LIN {X 0,Y 389.238,Z 288.654,A -85,B 0,C 180,E1 -14313.105,E2 -14313.105} C_VEL
LIN {X 0,Y 387.614,Z 288.058,A -85,B 0,C 180,E1 -14314.941,E2 -14314.941} C_VEL
LIN {X 0,Y 385.469,Z 286.733,A -85,B 0,C 180,E1 -14316.684,E2 -14316.684} C_VEL
LIN {X 0,Y 383.225,Z 284.713,A -85,B 0,C 180,E1 -14318.163,E2 -14318.163} C_VEL
LIN {X 0,Y 380.545,Z 281.669,A -85,B 0,C 180,E1 -14319.669,E2 -14319.669} C_VEL
LIN {X 0,Y 377.534,Z 279.906,A -85,B 0,C 180,E1 -14321.039,E2 -14321.039} C_VEL
LIN {X 0,Y 374.063,Z 276.681,A -85,B 0,C 180,E1 -14322.478,E2 -14322.478} C_VEL
LIN {X 0,Y 371.999,Z 274.442,A -85,B 0,C 180,E1 -14323.274,E2 -14323.274} C_VEL
LIN {X 0,Y 368.238,Z 271.447,A -85,B 0,C 180,E1 -14324.55,E2 -14324.55} C_VEL
LIN {X 0,Y 365.07,Z 267.86,A -85,B 0,C 180,E1 -14325.587,E2 -14325.587} C_VEL
LIN {X 0,Y 361.353,Z 264.675,A -85,B 0,C 180,E1 -14326.692,E2 -14326.692} C_VEL
LIN {X 0,Y 358.552,Z 261.44,A -85,B 0,C 180,E1 -14327.482,E2 -14327.482} C_VEL
LIN {X 0,Y 355.376,Z 258.454,A -85,B 0,C 180,E1 -14328.333,E2 -14328.333} C_VEL
LIN {X 0,Y 353.051,Z 255.522,A -85,B 0,C 180,E1 -14328.94,E2 -14328.94} C_VEL
LIN {X 0,Y 350.001,Z 252.371,A -85,B 0,C 180,E1 -14329.706,E2 -14329.706} C_VEL
LIN {X 0,Y 348.215,Z 249.968,A -85,B 0,C 180,E1 -14330.137,E2 -14330.137} C_VEL
LIN {X 0,Y 345.498,Z 247.058,A -85,B 0,C 180,E1 -14330.785,E2 -14330.785} C_VEL
LIN {X 0,Y 344.015,Z 244.683,A -85,B 0,C 180,E1 -14331.145,E2 -14331.145} C_VEL
LIN {X 0,Y 341.721,Z 242.357,A -85,B 0,C 180,E1 -14331.634,E2 -14331.634} C_VEL
LIN {X 0,Y 340.82,Z 240.079,A -85,B 0,C 180,E1 -14331.984,E2 -14331.984} C_VEL
LIN {X 0,Y 340.743,Z 239.555,A -85,B 0,C 180,E1 -14332.43,E2 -14332.43} C_VEL
LIN {X 0,Y 340.769,Z 239.539,A -85,B 0,C 180,E1 -14335.665,E2 -14335.665} C_VEL
LIN {X 0,Y 340.724,Z 239.527,A -85,B 0,C 180,E1 -14338.321,E2 -14338.321} C_VEL
LIN {X 0,Y 340.694,Z 239.543,A -85,B 0,C 180,E1 -14341.045,E2 -14341.045} C_VEL
LIN {X 0,Y 340.714,Z 239.518,A -85,B 0,C 180,E1 -14345.279,E2 -14345.279} C_VEL
LIN {X 0,Y 340.714,Z 239.545,A -85,B 0,C 180,E1 -14348.388,E2 -14348.388} C_VEL
LIN {X 0,Y 340.702,Z 239.5,A -85,B 0,C 180,E1 -14352.047,E2 -14352.047} C_VEL
LIN {X 0,Y 340.751,Z 239.541,A -85,B 0,C 180,E1 -14356.209,E2 -14356.209} C_VEL
LIN {X 0,Y 340.761,Z 239.524,A -85,B 0,C 180,E1 -14359.738,E2 -14359.738} C_VEL
LIN {X 0,Y 340.708,Z 239.542,A -85,B 0,C 180,E1 -14363.56,E2 -14363.56} C_VEL
LIN {X 0,Y 340.689,Z 239.532,A -85,B 0,C 180,E1 -14366.154,E2 -14366.154} C_VEL
LIN {X 0,Y 340.772,Z 239.531,A -85,B 0,C 180,E1 -14370.333,E2 -14370.333} C_VEL
LIN {X 0,Y 340.801,Z 239.508,A -85,B 0,C 180,E1 -14373.021,E2 -14373.021} C_VEL
LIN {X 0,Y 340.758,Z 239.53,A -85,B 0,C 180,E1 -14374.684,E2 -14374.684} C_VEL
LIN {X 0,Y 340.074,Z 239.623,A -85,B 0,C 180,E1 -14375.671,E2 -14375.671} C_VEL
LIN {X 0,Y 337.177,Z 239.985,A -85,B 0,C 180,E1 -14377.275,E2 -14377.275} C_VEL
LIN {X 0,Y 334.754,Z 240.278,A -85,B 0,C 180,E1 -14378.574,E2 -14378.574} C_VEL
LIN {X 0,Y 333.754,Z 240.389,A -85,B 0,C 180,E1 -14379.58,E2 -14379.58} C_VEL
LIN {X 0,Y 333.694,Z 240.393,A -85,B 0,C 180,E1 -14379.921,E2 -14379.921} C_VEL
LIN {X 0,Y 333.745,Z 240.399,A -85,B 0,C 180,E1 -14382.854,E2 -14382.854} C_VEL
LIN {X 0,Y 333.795,Z 240.402,A -85,B 0,C 180,E1 -14386.609,E2 -14386.609} C_VEL
LIN {X 0,Y 333.849,Z 240.365,A -85,B 0,C 180,E1 -14390.305,E2 -14390.305} C_VEL
LIN {X 0,Y 334.004,Z 240.369,A -85,B 0,C 180,E1 -14392.748,E2 -14392.748} C_VEL
LIN {X 0,Y 333.808,Z 240.407,A -85,B 0,C 180,E1 -14395.17,E2 -14395.17} C_VEL
LIN {X 0,Y 334.106,Z 240.351,A -85,B 0,C 180,E1 -14397.589,E2 -14397.589} C_VEL
LIN {X 0,Y 334.226,Z 240.318,A -85,B 0,C 180,E1 -14400.001,E2 -14400.001} C_VEL
LIN {X 0,Y 334.105,Z 240.356,A -85,B 0,C 180,E1 -14402.412,E2 -14402.412} C_VEL
LIN {X 0,Y 333.998,Z 240.376,A -85,B 0,C 180,E1 -14406.04,E2 -14406.04} C_VEL
LIN {X 0,Y 333.82,Z 240.368,A -85,B 0,C 180,E1 -14409.697,E2 -14409.697} C_VEL
LIN {X 0,Y 333.797,Z 240.403,A -85,B 0,C 180,E1 -14413.392,E2 -14413.392} C_VEL
LIN {X 0,Y 333.719,Z 240.394,A -85,B 0,C 180,E1 -14417.148,E2 -14417.148} C_VEL
LIN {X 0,Y 333.719,Z 240.392,A -85,B 0,C 180,E1 -14419.692,E2 -14419.692} C_VEL
LIN {X 0,Y 333.692,Z 240.415,A -85,B 0,C 180,E1 -14422.279,E2 -14422.279} C_VEL
LIN {X 0,Y 333.735,Z 240.391,A -85,B 0,C 180,E1 -14426.247,E2 -14426.247} C_VEL
LIN {X 0,Y 333.691,Z 240.412,A -85,B 0,C 180,E1 -14428.975,E2 -14428.975} C_VEL
LIN {X 0,Y 333.644,Z 240.414,A -85,B 0,C 180,E1 -14432.587,E2 -14432.587} C_VEL
LIN {X 0,Y 333.675,Z 240.415,A -85,B 0,C 180,E1 -14436.14,E2 -14436.14} C_VEL
LIN {X 0,Y 333.648,Z 240.414,A -85,B 0,C 180,E1 -14439.193,E2 -14439.193} C_VEL
LIN {X 0,Y 333.634,Z 240.428,A -85,B 0,C 180,E1 -14442.501,E2 -14442.501} C_VEL
LIN {X 0,Y 333.598,Z 240.43,A -85,B 0,C 180,E1 -14445.956,E2 -14445.956} C_VEL
LIN {X 0,Y 333.649,Z 240.398,A -85,B 0,C 180,E1 -14449.316,E2 -14449.316} C_VEL
LIN {X 0,Y 333.667,Z 240.415,A -85,B 0,C 180,E1 -14453.168,E2 -14453.168} C_VEL
LIN {X 0,Y 333.701,Z 240.526,A -85,B 0,C 180,E1 -14456.885,E2 -14456.885} C_VEL
LIN {X 0,Y 335.005,Z 246.874,A -85,B 0,C 180,E1 -14459.332,E2 -14459.332} C_VEL
LIN {X 0,Y 336.843,Z 256.44,A -85,B 0,C 180,E1 -14462.677,E2 -14462.677} C_VEL
LIN {X 0,Y 337.125,Z 259.361,A -85,B 0,C 180,E1 -14463.692,E2 -14463.692} C_VEL
LIN {X 0,Y 336.268,Z 266.228,A -85,B 0,C 180,E1 -14465.913,E2 -14465.913} C_VEL
LIN {X 0,Y 336.94,Z 270.047,A -85,B 0,C 180,E1 -14466.119,E2 -14466.119} C_VEL
LIN {X 0,Y 341.597,Z 292.634,A -85,B 0,C 180,E1 -14466.967,E2 -14466.967} C_VEL
LIN {X 0,Y 343.681,Z 305.633,A -85,B 0,C 180,E1 -14467.402,E2 -14467.402} C_VEL
LIN {X 0,Y 342.412,Z 371.156,A -85,B 0,C 180,E1 -14468.792,E2 -14468.792} C_VEL
LIN {X 0,Y 341.886,Z 381.9,A -85,B 0,C 180,E1 -14469.152,E2 -14469.152} C_VEL
LIN {X 0,Y 341.255,Z 391.001,A -85,B 0,C 180,E1 -14469.585,E2 -14469.585} C_VEL
LIN {X 0,Y 340.336,Z 401.361,A -85,B 0,C 180,E1 -14470.236,E2 -14470.236} C_VEL
LIN {X 0,Y 339.44,Z 410.495,A -85,B 0,C 180,E1 -14470.968,E2 -14470.968} C_VEL
LIN {X 0,Y 338.419,Z 419.49,A -85,B 0,C 180,E1 -14471.85,E2 -14471.85} C_VEL
LIN {X 0,Y 337.282,Z 428.216,A -85,B 0,C 180,E1 -14472.883,E2 -14472.883} C_VEL
LIN {X 0,Y 336.343,Z 435.977,A -85,B 0,C 180,E1 -14473.986,E2 -14473.986} C_VEL
LIN {X 0,Y 335.454,Z 442.832,A -85,B 0,C 180,E1 -14475.129,E2 -14475.129} C_VEL
LIN {X 0,Y 334.667,Z 449.035,A -85,B 0,C 180,E1 -14476.335,E2 -14476.335} C_VEL
LIN {X 0,Y 333.732,Z 455.57,A -85,B 0,C 180,E1 -14477.843,E2 -14477.843} C_VEL
LIN {X 0,Y 333.236,Z 460.074,A -85,B 0,C 180,E1 -14479.058,E2 -14479.058} C_VEL
LIN {X 0,Y 332.605,Z 465.566,A -85,B 0,C 180,E1 -14480.882,E2 -14480.882} C_VEL
LIN {X 0,Y 332.202,Z 469.891,A -85,B 0,C 180,E1 -14482.708,E2 -14482.708} C_VEL
LIN {X 0,Y 332.034,Z 472.629,A -85,B 0,C 180,E1 -14484.174,E2 -14484.174} C_VEL
LIN {X 0,Y 331.97,Z 475.448,A -85,B 0,C 180,E1 -14486.359,E2 -14486.359} C_VEL
LIN {X 0,Y 331.916,Z 476.506,A -85,B 0,C 180,E1 -14487.573,E2 -14487.573} C_VEL
LIN {X 0,Y 331.913,Z 477.095,A -85,B 0,C 180,E1 -14488.787,E2 -14488.787} C_VEL
LIN {X 0,Y 331.913,Z 477.095,A -85,B 0,C 180,E1 -14491.213,E2 -14491.213} C_VEL
LIN {X 0,Y 331.916,Z 476.506,A -85,B 0,C 180,E1 -14492.427,E2 -14492.427} C_VEL
LIN {X 0,Y 331.971,Z 474.059,A -85,B 0,C 180,E1 -14494.858,E2 -14494.858} C_VEL
LIN {X 0,Y 332.105,Z 471.109,A -85,B 0,C 180,E1 -14496.684,E2 -14496.684} C_VEL
LIN {X 0,Y 332.461,Z 467.12,A -85,B 0,C 180,E1 -14498.51,E2 -14498.51} C_VEL
LIN {X 0,Y 332.985,Z 461.99,A -85,B 0,C 180,E1 -14500.335,E2 -14500.335} C_VEL
LIN {X 0,Y 333.589,Z 456.726,A -85,B 0,C 180,E1 -14501.854,E2 -14501.854} C_VEL
LIN {X 0,Y 334.455,Z 450.41,A -85,B 0,C 180,E1 -14503.364,E2 -14503.364} C_VEL
LIN {X 0,Y 335.208,Z 444.458,A -85,B 0,C 180,E1 -14504.572,E2 -14504.572} C_VEL
LIN {X 0,Y 336.147,Z 437.531,A -85,B 0,C 180,E1 -14505.771,E2 -14505.771} C_VEL
LIN {X 0,Y 337.155,Z 429.351,A -85,B 0,C 180,E1 -14506.967,E2 -14506.967} C_VEL
LIN {X 0,Y 338.249,Z 420.841,A -85,B 0,C 180,E1 -14508.003,E2 -14508.003} C_VEL
LIN {X 0,Y 339.26,Z 412.127,A -85,B 0,C 180,E1 -14508.886,E2 -14508.886} C_VEL
LIN {X 0,Y 340.256,Z 402.369,A -85,B 0,C 180,E1 -14509.69,E2 -14509.69} C_VEL
LIN {X 0,Y 341.184,Z 392.289,A -85,B 0,C 180,E1 -14510.341,E2 -14510.341} C_VEL
LIN {X 0,Y 341.848,Z 382.775,A -85,B 0,C 180,E1 -14510.811,E2 -14510.811} C_VEL
LIN {X 0,Y 342.38,Z 372.463,A -85,B 0,C 180,E1 -14511.17,E2 -14511.17} C_VEL
LIN {X 0,Y 343.694,Z 305.784,A -85,B 0,C 180,E1 -14512.594,E2 -14512.594} C_VEL
LIN {X 0,Y 339.925,Z 283.944,A -85,B 0,C 180,E1 -14513.347,E2 -14513.347} C_VEL
LIN {X 0,Y 336.278,Z 266.684,A -85,B 0,C 180,E1 -14514.03,E2 -14514.03} C_VEL
LIN {X 0,Y 336.36,Z 265.08,A -85,B 0,C 180,E1 -14514.405,E2 -14514.405} C_VEL
LIN {X 0,Y 337.108,Z 259.382,A -85,B 0,C 180,E1 -14516.302,E2 -14516.302} C_VEL
LIN {X 0,Y 336.549,Z 254.647,A -85,B 0,C 180,E1 -14517.961,E2 -14517.961} C_VEL
LIN {X 0,Y 334.535,Z 244.335,A -85,B 0,C 180,E1 -14521.682,E2 -14521.682} C_VEL
LIN {X 0,Y 333.674,Z 240.436,A -85,B 0,C 180,E1 -14523.204,E2 -14523.204} C_VEL
LIN {X 0,Y 333.667,Z 240.415,A -85,B 0,C 180,E1 -14526.832,E2 -14526.832} C_VEL
LIN {X 0,Y 333.648,Z 240.398,A -85,B 0,C 180,E1 -14530.767,E2 -14530.767} C_VEL
LIN {X 0,Y 333.595,Z 240.428,A -85,B 0,C 180,E1 -14534.25,E2 -14534.25} C_VEL
LIN {X 0,Y 333.643,Z 240.428,A -85,B 0,C 180,E1 -14537.618,E2 -14537.618} C_VEL
LIN {X 0,Y 333.653,Z 240.416,A -85,B 0,C 180,E1 -14541.202,E2 -14541.202} C_VEL
LIN {X 0,Y 333.675,Z 240.415,A -85,B 0,C 180,E1 -14543.86,E2 -14543.86} C_VEL
LIN {X 0,Y 333.644,Z 240.414,A -85,B 0,C 180,E1 -14547.413,E2 -14547.413} C_VEL
LIN {X 0,Y 333.691,Z 240.412,A -85,B 0,C 180,E1 -14551.025,E2 -14551.025} C_VEL
LIN {X 0,Y 333.735,Z 240.391,A -85,B 0,C 180,E1 -14553.753,E2 -14553.753} C_VEL
LIN {X 0,Y 333.72,Z 240.41,A -85,B 0,C 180,E1 -14557.913,E2 -14557.913} C_VEL
LIN {X 0,Y 333.741,Z 240.382,A -85,B 0,C 180,E1 -14561.586,E2 -14561.586} C_VEL
LIN {X 0,Y 333.808,Z 240.402,A -85,B 0,C 180,E1 -14565.576,E2 -14565.576} C_VEL
LIN {X 0,Y 333.817,Z 240.377,A -85,B 0,C 180,E1 -14569.077,E2 -14569.077} C_VEL
LIN {X 0,Y 333.968,Z 240.369,A -85,B 0,C 180,E1 -14572.746,E2 -14572.746} C_VEL
LIN {X 0,Y 333.804,Z 240.406,A -85,B 0,C 180,E1 -14575.168,E2 -14575.168} C_VEL
LIN {X 0,Y 334.105,Z 240.356,A -85,B 0,C 180,E1 -14577.588,E2 -14577.588} C_VEL
LIN {X 0,Y 334.226,Z 240.318,A -85,B 0,C 180,E1 -14579.999,E2 -14579.999} C_VEL
LIN {X 0,Y 334.106,Z 240.351,A -85,B 0,C 180,E1 -14582.411,E2 -14582.411} C_VEL
LIN {X 0,Y 333.99,Z 240.374,A -85,B 0,C 180,E1 -14586.597,E2 -14586.597} C_VEL
LIN {X 0,Y 333.849,Z 240.365,A -85,B 0,C 180,E1 -14589.695,E2 -14589.695} C_VEL
LIN {X 0,Y 333.795,Z 240.402,A -85,B 0,C 180,E1 -14593.391,E2 -14593.391} C_VEL
LIN {X 0,Y 333.745,Z 240.399,A -85,B 0,C 180,E1 -14597.146,E2 -14597.146} C_VEL
LIN {X 0,Y 333.729,Z 240.386,A -85,B 0,C 180,E1 -14599.69,E2 -14599.69} C_VEL
LIN {X 0,Y 333.667,Z 240.421,A -85,B 0,C 180,E1 -14603.59,E2 -14603.59} C_VEL
LIN {X 0,Y 333.732,Z 240.394,A -85,B 0,C 180,E1 -14606.246,E2 -14606.246} C_VEL
LIN {X 0,Y 333.708,Z 240.407,A -85,B 0,C 180,E1 -14608.972,E2 -14608.972} C_VEL
LIN {X 0,Y 333.64,Z 240.419,A -85,B 0,C 180,E1 -14612.586,E2 -14612.586} C_VEL
LIN {X 0,Y 333.673,Z 240.413,A -85,B 0,C 180,E1 -14616.138,E2 -14616.138} C_VEL
LIN {X 0,Y 333.679,Z 240.417,A -85,B 0,C 180,E1 -14619.187,E2 -14619.187} C_VEL
LIN {X 0,Y 333.7,Z 240.418,A -85,B 0,C 180,E1 -14622.513,E2 -14622.513} C_VEL
LIN {X 0,Y 333.631,Z 240.402,A -85,B 0,C 180,E1 -14625.961,E2 -14625.961} C_VEL
LIN {X 0,Y 333.651,Z 240.389,A -85,B 0,C 180,E1 -14629.314,E2 -14629.314} C_VEL
LIN {X 0,Y 333.652,Z 240.424,A -85,B 0,C 180,E1 -14632.349,E2 -14632.349} C_VEL
LIN {X 0,Y 333.67,Z 240.392,A -85,B 0,C 180,E1 -14635.341,E2 -14635.341} C_VEL
LIN {X 0,Y 333.686,Z 240.404,A -85,B 0,C 180,E1 -14639.637,E2 -14639.637} C_VEL
LIN {X 0,Y 333.736,Z 240.41,A -85,B 0,C 180,E1 -14642.401,E2 -14642.401} C_VEL
LIN {X 0,Y 333.723,Z 240.417,A -85,B 0,C 180,E1 -14645.091,E2 -14645.091} C_VEL
LIN {X 0,Y 333.714,Z 240.563,A -85,B 0,C 180,E1 -14646.635,E2 -14646.635} C_VEL
LIN {X 0,Y 333.902,Z 241.475,A -85,B 0,C 180,E1 -14646.906,E2 -14646.906} C_VEL
LIN {X 0,Y 335.441,Z 244.25,A -85,B 0,C 180,E1 -14647.293,E2 -14647.293} C_VEL
LIN {X 0,Y 337.24,Z 246.138,A -85,B 0,C 180,E1 -14647.649,E2 -14647.649} C_VEL
LIN {X 0,Y 339.606,Z 249.544,A -85,B 0,C 180,E1 -14648.193,E2 -14648.193} C_VEL
LIN {X 0,Y 341.244,Z 251.3,A -85,B 0,C 180,E1 -14648.55,E2 -14648.55} C_VEL
LIN {X 0,Y 344.183,Z 255.015,A -85,B 0,C 180,E1 -14649.205,E2 -14649.205} C_VEL
LIN {X 0,Y 346.131,Z 257.085,A -85,B 0,C 180,E1 -14649.669,E2 -14649.669} C_VEL
LIN {X 0,Y 349.255,Z 260.734,A -85,B 0,C 180,E1 -14650.409,E2 -14650.409} C_VEL
LIN {X 0,Y 351.306,Z 262.788,A -85,B 0,C 180,E1 -14650.915,E2 -14650.915} C_VEL
LIN {X 0,Y 354.984,Z 266.845,A -85,B 0,C 180,E1 -14651.859,E2 -14651.859} C_VEL
LIN {X 0,Y 357.12,Z 268.84,A -85,B 0,C 180,E1 -14652.431,E2 -14652.431} C_VEL
LIN {X 0,Y 361.088,Z 272.942,A -85,B 0,C 180,E1 -14653.544,E2 -14653.544} C_VEL
LIN {X 0,Y 363.916,Z 275.38,A -85,B 0,C 180,E1 -14654.391,E2 -14654.391} C_VEL
LIN {X 0,Y 367.522,Z 279.123,A -85,B 0,C 180,E1 -14655.553,E2 -14655.553} C_VEL
LIN {X 0,Y 371.229,Z 282.06,A -85,B 0,C 180,E1 -14656.813,E2 -14656.813} C_VEL
LIN {X 0,Y 374.888,Z 285.747,A -85,B 0,C 180,E1 -14658.242,E2 -14658.242} C_VEL
LIN {X 0,Y 378.477,Z 288.218,A -85,B 0,C 180,E1 -14659.786,E2 -14659.786} C_VEL
LIN {X 0,Y 379.883,Z 289.155,A -85,B 0,C 180,E1 -14660.464,E2 -14660.464} C_VEL
LIN {X 0,Y 382.521,Z 292.118,A -85,B 0,C 180,E1 -14661.961,E2 -14661.961} C_VEL
LIN {X 0,Y 384.968,Z 294.058,A -85,B 0,C 180,E1 -14663.58,E2 -14663.58} C_VEL
LIN {X 0,Y 387.283,Z 295.335,A -85,B 0,C 180,E1 -14665.578,E2 -14665.578} C_VEL
LIN {X 0,Y 388.665,Z 295.823,A -85,B 0,C 180,E1 -14667.428,E2 -14667.428} C_VEL
LIN {X 0,Y 389.239,Z 296.26,A -85,B 0,C 180,E1 -14668.965,E2 -14668.965} C_VEL
LIN {X 0,Y 389.407,Z 296.18,A -85,B 0,C 180,E1 -14670,E2 -14670} C_VEL
LIN {X 0,Y 389.127,Z 296.134,A -85,B 0,C 180,E1 -14671.552,E2 -14671.552} C_VEL
LIN {X 0,Y 388.361,Z 295.7,A -85,B 0,C 180,E1 -14673.112,E2 -14673.112} C_VEL
LIN {X 0,Y 386.736,Z 295.097,A -85,B 0,C 180,E1 -14674.943,E2 -14674.943} C_VEL
LIN {X 0,Y 384.56,Z 293.784,A -85,B 0,C 180,E1 -14676.7,E2 -14676.7} C_VEL
LIN {X 0,Y 382.221,Z 291.835,A -85,B 0,C 180,E1 -14678.214,E2 -14678.214} C_VEL
LIN {X 0,Y 379.213,Z 288.562,A -85,B 0,C 180,E1 -14679.864,E2 -14679.864} C_VEL
LIN {X 0,Y 376.134,Z 286.754,A -85,B 0,C 180,E1 -14681.228,E2 -14681.228} C_VEL
LIN {X 0,Y 372.666,Z 283.664,A -85,B 0,C 180,E1 -14682.629,E2 -14682.629} C_VEL
LIN {X 0,Y 370.003,Z 280.944,A -85,B 0,C 180,E1 -14683.635,E2 -14683.635} C_VEL
LIN {X 0,Y 365.739,Z 277.428,A -85,B 0,C 180,E1 -14685.039,E2 -14685.039} C_VEL
LIN {X 0,Y 362.686,Z 274.176,A -85,B 0,C 180,E1 -14685.985,E2 -14685.985} C_VEL
LIN {X 0,Y 358.817,Z 270.811,A -85,B 0,C 180,E1 -14687.085,E2 -14687.085} C_VEL
LIN {X 0,Y 355.813,Z 267.509,A -85,B 0,C 180,E1 -14687.929,E2 -14687.929} C_VEL
LIN {X 0,Y 352.189,Z 263.983,A -85,B 0,C 180,E1 -14688.848,E2 -14688.848} C_VEL
LIN {X 0,Y 350.012,Z 261.386,A -85,B 0,C 180,E1 -14689.415,E2 -14689.415} C_VEL
LIN {X 0,Y 346.374,Z 257.473,A -85,B 0,C 180,E1 -14690.27,E2 -14690.27} C_VEL
LIN {X 0,Y 344.964,Z 255.745,A -85,B 0,C 180,E1 -14690.614,E2 -14690.614} C_VEL
LIN {X 0,Y 341.952,Z 252.422,A -85,B 0,C 180,E1 -14691.286,E2 -14691.286} C_VEL
LIN {X 0,Y 340.284,Z 250.185,A -85,B 0,C 180,E1 -14691.661,E2 -14691.661} C_VEL
LIN {X 0,Y 337.761,Z 247.052,A -85,B 0,C 180,E1 -14692.231,E2 -14692.231} C_VEL
LIN {X 0,Y 336.543,Z 245.281,A -85,B 0,C 180,E1 -14692.493,E2 -14692.493} C_VEL
LIN {X 0,Y 334.617,Z 243.125,A -85,B 0,C 180,E1 -14692.878,E2 -14692.878} C_VEL
LIN {X 0,Y 333.802,Z 241.07,A -85,B 0,C 180,E1 -14693.171,E2 -14693.171} C_VEL
LIN {X 0,Y 333.68,Z 240.493,A -85,B 0,C 180,E1 -14693.425,E2 -14693.425} C_VEL
LIN {X 0,Y 333.731,Z 240.416,A -85,B 0,C 180,E1 -14696.247,E2 -14696.247} C_VEL
LIN {X 0,Y 333.686,Z 240.398,A -85,B 0,C 180,E1 -14698.974,E2 -14698.974} C_VEL
LIN {X 0,Y 333.639,Z 240.42,A -85,B 0,C 180,E1 -14702.587,E2 -14702.587} C_VEL
LIN {X 0,Y 333.673,Z 240.405,A -85,B 0,C 180,E1 -14706.139,E2 -14706.139} C_VEL
LIN {X 0,Y 333.668,Z 240.416,A -85,B 0,C 180,E1 -14709.189,E2 -14709.189} C_VEL
LIN {X 0,Y 333.635,Z 240.381,A -85,B 0,C 180,E1 -14712.501,E2 -14712.501} C_VEL
LIN {X 0,Y 333.697,Z 240.417,A -85,B 0,C 180,E1 -14715.973,E2 -14715.973} C_VEL
LIN {X 0,Y 333.699,Z 240.402,A -85,B 0,C 180,E1 -14719.305,E2 -14719.305} C_VEL
LIN {X 0,Y 333.663,Z 240.422,A -85,B 0,C 180,E1 -14723.168,E2 -14723.168} C_VEL
LIN {X 0,Y 333.671,Z 240.403,A -85,B 0,C 180,E1 -14725.342,E2 -14725.342} C_VEL
LIN {X 0,Y 333.7,Z 240.418,A -85,B 0,C 180,E1 -14729.711,E2 -14729.711} C_VEL
LIN {X 0,Y 333.739,Z 240.387,A -85,B 0,C 180,E1 -14732.402,E2 -14732.402} C_VEL
LIN {X 0,Y 333.723,Z 240.408,A -85,B 0,C 180,E1 -14735.091,E2 -14735.091} C_VEL
LIN {X 0,Y 333.671,Z 240.409,A -85,B 0,C 180,E1 -14739.019,E2 -14739.019} C_VEL
LIN {X 0,Y 333.694,Z 240.393,A -85,B 0,C 180,E1 -14739.921,E2 -14739.921} C_VEL
LIN {X 0,Y 333.085,Z 240.467,A -85,B 0,C 180,E1 -14740.928,E2 -14740.928} C_VEL
LIN {X 0,Y 330.264,Z 240.832,A -85,B 0,C 180,E1 -14742.567,E2 -14742.567} C_VEL
LIN {X 0,Y 327.851,Z 241.144,A -85,B 0,C 180,E1 -14743.895,E2 -14743.895} C_VEL
LIN {X 0,Y 326.829,Z 241.272,A -85,B 0,C 180,E1 -14744.923,E2 -14744.923} C_VEL
LIN {X 0,Y 326.756,Z 241.284,A -85,B 0,C 180,E1 -14745.271,E2 -14745.271} C_VEL
LIN {X 0,Y 326.768,Z 241.256,A -85,B 0,C 180,E1 -14748.84,E2 -14748.84} C_VEL
LIN {X 0,Y 326.957,Z 241.246,A -85,B 0,C 180,E1 -14752.591,E2 -14752.591} C_VEL
LIN {X 0,Y 326.775,Z 241.282,A -85,B 0,C 180,E1 -14755.066,E2 -14755.066} C_VEL
LIN {X 0,Y 327.046,Z 241.23,A -85,B 0,C 180,E1 -14757.537,E2 -14757.537} C_VEL
LIN {X 0,Y 327.178,Z 241.195,A -85,B 0,C 180,E1 -14760.001,E2 -14760.001} C_VEL
LIN {X 0,Y 327.045,Z 241.236,A -85,B 0,C 180,E1 -14762.464,E2 -14762.464} C_VEL
LIN {X 0,Y 326.952,Z 241.254,A -85,B 0,C 180,E1 -14766.171,E2 -14766.171} C_VEL
LIN {X 0,Y 326.783,Z 241.245,A -85,B 0,C 180,E1 -14769.908,E2 -14769.908} C_VEL
LIN {X 0,Y 326.759,Z 241.278,A -85,B 0,C 180,E1 -14773.686,E2 -14773.686} C_VEL
LIN {X 0,Y 326.664,Z 241.269,A -85,B 0,C 180,E1 -14777.531,E2 -14777.531} C_VEL
LIN {X 0,Y 326.653,Z 241.276,A -85,B 0,C 180,E1 -14780.136,E2 -14780.136} C_VEL
LIN {X 0,Y 326.651,Z 241.293,A -85,B 0,C 180,E1 -14784.13,E2 -14784.13} C_VEL
LIN {X 0,Y 326.683,Z 241.267,A -85,B 0,C 180,E1 -14786.858,E2 -14786.858} C_VEL
LIN {X 0,Y 326.635,Z 241.301,A -85,B 0,C 180,E1 -14790.61,E2 -14790.61} C_VEL
LIN {X 0,Y 326.607,Z 241.281,A -85,B 0,C 180,E1 -14794.02,E2 -14794.02} C_VEL
LIN {X 0,Y 326.627,Z 241.298,A -85,B 0,C 180,E1 -14797.239,E2 -14797.239} C_VEL
LIN {X 0,Y 326.579,Z 241.3,A -85,B 0,C 180,E1 -14801.132,E2 -14801.132} C_VEL
LIN {X 0,Y 326.529,Z 241.304,A -85,B 0,C 180,E1 -14804.743,E2 -14804.743} C_VEL
LIN {X 0,Y 326.578,Z 241.29,A -85,B 0,C 180,E1 -14808.155,E2 -14808.155} C_VEL
LIN {X 0,Y 326.626,Z 241.292,A -85,B 0,C 180,E1 -14811.392,E2 -14811.392} C_VEL
LIN {X 0,Y 326.621,Z 241.285,A -85,B 0,C 180,E1 -14814.852,E2 -14814.852} C_VEL
LIN {X 0,Y 326.638,Z 241.442,A -85,B 0,C 180,E1 -14816.485,E2 -14816.485} C_VEL
LIN {X 0,Y 328.254,Z 249.049,A -85,B 0,C 180,E1 -14819.437,E2 -14819.437} C_VEL
LIN {X 0,Y 329.631,Z 256.233,A -85,B 0,C 180,E1 -14822.027,E2 -14822.027} C_VEL
LIN {X 0,Y 330.178,Z 260.185,A -85,B 0,C 180,E1 -14823.449,E2 -14823.449} C_VEL
LIN {X 0,Y 329.441,Z 266.047,A -85,B 0,C 180,E1 -14825.384,E2 -14825.384} C_VEL
LIN {X 0,Y 330.28,Z 270.396,A -85,B 0,C 180,E1 -14825.62,E2 -14825.62} C_VEL
LIN {X 0,Y 335.118,Z 293.847,A -85,B 0,C 180,E1 -14826.528,E2 -14826.528} C_VEL
LIN {X 0,Y 337.12,Z 306.638,A -85,B 0,C 180,E1 -14826.964,E2 -14826.964} C_VEL
LIN {X 0,Y 335.787,Z 372.27,A -85,B 0,C 180,E1 -14828.393,E2 -14828.393} C_VEL
LIN {X 0,Y 335.205,Z 382.582,A -85,B 0,C 180,E1 -14828.757,E2 -14828.757} C_VEL
LIN {X 0,Y 334.495,Z 392.095,A -85,B 0,C 180,E1 -14829.234,E2 -14829.234} C_VEL
LIN {X 0,Y 333.669,Z 401.169,A -85,B 0,C 180,E1 -14829.824,E2 -14829.824} C_VEL
LIN {X 0,Y 332.729,Z 410.302,A -85,B 0,C 180,E1 -14830.569,E2 -14830.569} C_VEL
LIN {X 0,Y 331.671,Z 419.297,A -85,B 0,C 180,E1 -14831.467,E2 -14831.467} C_VEL
LIN {X 0,Y 330.485,Z 428.023,A -85,B 0,C 180,E1 -14832.52,E2 -14832.52} C_VEL
LIN {X 0,Y 329.543,Z 435.422,A -85,B 0,C 180,E1 -14833.587,E2 -14833.587} C_VEL
LIN {X 0,Y 328.573,Z 442.685,A -85,B 0,C 180,E1 -14834.819,E2 -14834.819} C_VEL
LIN {X 0,Y 327.76,Z 448.842,A -85,B 0,C 180,E1 -14836.041,E2 -14836.041} C_VEL
LIN {X 0,Y 326.768,Z 455.377,A -85,B 0,C 180,E1 -14837.58,E2 -14837.58} C_VEL
LIN {X 0,Y 326.212,Z 459.88,A -85,B 0,C 180,E1 -14838.82,E2 -14838.82} C_VEL
LIN {X 0,Y 325.573,Z 465.373,A -85,B 0,C 180,E1 -14840.683,E2 -14840.683} C_VEL
LIN {X 0,Y 325.153,Z 469.699,A -85,B 0,C 180,E1 -14842.549,E2 -14842.549} C_VEL
LIN {X 0,Y 324.925,Z 472.731,A -85,B 0,C 180,E1 -14844.251,E2 -14844.251} C_VEL
LIN {X 0,Y 324.876,Z 475.255,A -85,B 0,C 180,E1 -14846.279,E2 -14846.279} C_VEL
LIN {X 0,Y 324.835,Z 476.314,A -85,B 0,C 180,E1 -14847.52,E2 -14847.52} C_VEL
LIN {X 0,Y 324.822,Z 476.903,A -85,B 0,C 180,E1 -14848.76,E2 -14848.76} C_VEL
LIN {X 0,Y 324.822,Z 476.903,A -85,B 0,C 180,E1 -14851.24,E2 -14851.24} C_VEL
LIN {X 0,Y 324.835,Z 476.314,A -85,B 0,C 180,E1 -14852.48,E2 -14852.48} C_VEL
LIN {X 0,Y 324.882,Z 473.866,A -85,B 0,C 180,E1 -14854.964,E2 -14854.964} C_VEL
LIN {X 0,Y 325.047,Z 470.916,A -85,B 0,C 180,E1 -14856.83,E2 -14856.83} C_VEL
LIN {X 0,Y 325.401,Z 466.927,A -85,B 0,C 180,E1 -14858.696,E2 -14858.696} C_VEL
LIN {X 0,Y 325.965,Z 461.796,A -85,B 0,C 180,E1 -14860.56,E2 -14860.56} C_VEL
LIN {X 0,Y 326.619,Z 456.533,A -85,B 0,C 180,E1 -14862.11,E2 -14862.11} C_VEL
LIN {X 0,Y 327.538,Z 450.217,A -85,B 0,C 180,E1 -14863.652,E2 -14863.652} C_VEL
LIN {X 0,Y 328.315,Z 444.264,A -85,B 0,C 180,E1 -14864.885,E2 -14864.885} C_VEL
LIN {X 0,Y 329.28,Z 437.338,A -85,B 0,C 180,E1 -14866.109,E2 -14866.109} C_VEL
LIN {X 0,Y 330.328,Z 429.157,A -85,B 0,C 180,E1 -14867.329,E2 -14867.329} C_VEL
LIN {X 0,Y 331.481,Z 420.648,A -85,B 0,C 180,E1 -14868.384,E2 -14868.384} C_VEL
LIN {X 0,Y 332.556,Z 411.934,A -85,B 0,C 180,E1 -14869.281,E2 -14869.281} C_VEL
LIN {X 0,Y 333.572,Z 402.176,A -85,B 0,C 180,E1 -14870.102,E2 -14870.102} C_VEL
LIN {X 0,Y 334.548,Z 392.097,A -85,B 0,C 180,E1 -14870.763,E2 -14870.763} C_VEL
LIN {X 0,Y 335.226,Z 382.582,A -85,B 0,C 180,E1 -14871.241,E2 -14871.241} C_VEL
LIN {X 0,Y 335.768,Z 372.27,A -85,B 0,C 180,E1 -14871.608,E2 -14871.608} C_VEL
LIN {X 0,Y 337.045,Z 305.805,A -85,B 0,C 180,E1 -14873.06,E2 -14873.06} C_VEL
LIN {X 0,Y 333.089,Z 283.374,A -85,B 0,C 180,E1 -14873.864,E2 -14873.864} C_VEL
LIN {X 0,Y 329.449,Z 266.337,A -85,B 0,C 180,E1 -14874.575,E2 -14874.575} C_VEL
LIN {X 0,Y 329.534,Z 264.885,A -85,B 0,C 180,E1 -14874.945,E2 -14874.945} C_VEL
LIN {X 0,Y 330.116,Z 260.063,A -85,B 0,C 180,E1 -14876.598,E2 -14876.598} C_VEL
LIN {X 0,Y 329.18,Z 253.676,A -85,B 0,C 180,E1 -14878.912,E2 -14878.912} C_VEL
LIN {X 0,Y 327.231,Z 244.125,A -85,B 0,C 180,E1 -14882.475,E2 -14882.475} C_VEL
LIN {X 0,Y 326.628,Z 241.356,A -85,B 0,C 180,E1 -14883.587,E2 -14883.587} C_VEL
LIN {X 0,Y 326.63,Z 241.297,A -85,B 0,C 180,E1 -14887.238,E2 -14887.238} C_VEL
LIN {X 0,Y 326.579,Z 241.28,A -85,B 0,C 180,E1 -14891.131,E2 -14891.131} C_VEL
LIN {X 0,Y 326.529,Z 241.306,A -85,B 0,C 180,E1 -14894.742,E2 -14894.742} C_VEL
LIN {X 0,Y 326.577,Z 241.303,A -85,B 0,C 180,E1 -14898.154,E2 -14898.154} C_VEL
LIN {X 0,Y 326.624,Z 241.293,A -85,B 0,C 180,E1 -14901.391,E2 -14901.391} C_VEL
LIN {X 0,Y 326.619,Z 241.287,A -85,B 0,C 180,E1 -14904.851,E2 -14904.851} C_VEL
LIN {X 0,Y 326.608,Z 241.291,A -85,B 0,C 180,E1 -14907.455,E2 -14907.455} C_VEL
LIN {X 0,Y 326.649,Z 241.293,A -85,B 0,C 180,E1 -14910.339,E2 -14910.339} C_VEL
LIN {X 0,Y 326.69,Z 241.275,A -85,B 0,C 180,E1 -14914.516,E2 -14914.516} C_VEL
LIN {X 0,Y 326.646,Z 241.291,A -85,B 0,C 180,E1 -14918.545,E2 -14918.545} C_VEL
LIN {X 0,Y 326.707,Z 241.258,A -85,B 0,C 180,E1 -14921.175,E2 -14921.175} C_VEL
LIN {X 0,Y 326.763,Z 241.28,A -85,B 0,C 180,E1 -14925.433,E2 -14925.433} C_VEL
LIN {X 0,Y 326.758,Z 241.258,A -85,B 0,C 180,E1 -14928.838,E2 -14928.838} C_VEL
LIN {X 0,Y 326.922,Z 241.245,A -85,B 0,C 180,E1 -14932.588,E2 -14932.588} C_VEL
LIN {X 0,Y 326.77,Z 241.283,A -85,B 0,C 180,E1 -14935.064,E2 -14935.064} C_VEL
LIN {X 0,Y 327.045,Z 241.236,A -85,B 0,C 180,E1 -14937.536,E2 -14937.536} C_VEL
LIN {X 0,Y 327.178,Z 241.195,A -85,B 0,C 180,E1 -14939.999,E2 -14939.999} C_VEL
LIN {X 0,Y 327.046,Z 241.23,A -85,B 0,C 180,E1 -14942.463,E2 -14942.463} C_VEL
LIN {X 0,Y 326.96,Z 241.251,A -85,B 0,C 180,E1 -14946.588,E2 -14946.588} C_VEL
LIN {X 0,Y 326.804,Z 241.242,A -85,B 0,C 180,E1 -14949.906,E2 -14949.906} C_VEL
LIN {X 0,Y 326.757,Z 241.279,A -85,B 0,C 180,E1 -14953.685,E2 -14953.685} C_VEL
LIN {X 0,Y 326.697,Z 241.274,A -85,B 0,C 180,E1 -14957.527,E2 -14957.527} C_VEL
LIN {X 0,Y 326.656,Z 241.27,A -85,B 0,C 180,E1 -14960.135,E2 -14960.135} C_VEL
LIN {X 0,Y 326.646,Z 241.297,A -85,B 0,C 180,E1 -14964.128,E2 -14964.128} C_VEL
LIN {X 0,Y 326.681,Z 241.266,A -85,B 0,C 180,E1 -14966.857,E2 -14966.857} C_VEL
LIN {X 0,Y 326.636,Z 241.299,A -85,B 0,C 180,E1 -14970.611,E2 -14970.611} C_VEL
LIN {X 0,Y 326.604,Z 241.284,A -85,B 0,C 180,E1 -14974.019,E2 -14974.019} C_VEL
LIN {X 0,Y 326.625,Z 241.298,A -85,B 0,C 180,E1 -14977.238,E2 -14977.238} C_VEL
LIN {X 0,Y 326.632,Z 241.284,A -85,B 0,C 180,E1 -14980.202,E2 -14980.202} C_VEL
LIN {X 0,Y 326.638,Z 241.298,A -85,B 0,C 180,E1 -14983.512,E2 -14983.512} C_VEL
LIN {X 0,Y 326.585,Z 241.262,A -85,B 0,C 180,E1 -14987.025,E2 -14987.025} C_VEL
LIN {X 0,Y 326.63,Z 241.291,A -85,B 0,C 180,E1 -14990.768,E2 -14990.768} C_VEL
LIN {X 0,Y 326.609,Z 241.275,A -85,B 0,C 180,E1 -14994.48,E2 -14994.48} C_VEL
LIN {X 0,Y 326.604,Z 241.297,A -85,B 0,C 180,E1 -14997.455,E2 -14997.455} C_VEL
LIN {X 0,Y 326.644,Z 241.275,A -85,B 0,C 180,E1 -15000.339,E2 -15000.339} C_VEL
LIN {X 0,Y 326.686,Z 241.293,A -85,B 0,C 180,E1 -15004.516,E2 -15004.516} C_VEL
LIN {X 0,Y 326.692,Z 241.587,A -85,B 0,C 180,E1 -15005.621,E2 -15005.621} C_VEL
LIN {X 0,Y 327.048,Z 242.916,A -85,B 0,C 180,E1 -15005.866,E2 -15005.866} C_VEL
LIN {X 0,Y 328.752,Z 245.549,A -85,B 0,C 180,E1 -15006.209,E2 -15006.209} C_VEL
LIN {X 0,Y 329.922,Z 246.856,A -85,B 0,C 180,E1 -15006.429,E2 -15006.429} C_VEL
LIN {X 0,Y 332.332,Z 250.357,A -85,B 0,C 180,E1 -15006.946,E2 -15006.946} C_VEL
LIN {X 0,Y 333.845,Z 252.169,A -85,B 0,C 180,E1 -15007.256,E2 -15007.256} C_VEL
LIN {X 0,Y 336.857,Z 255.833,A -85,B 0,C 180,E1 -15007.873,E2 -15007.873} C_VEL
LIN {X 0,Y 341.329,Z 261.193,A -85,B 0,C 180,E1 -15008.866,E2 -15008.866} C_VEL
LIN {X 0,Y 343.414,Z 263.466,A -85,B 0,C 180,E1 -15009.321,E2 -15009.321} C_VEL
LIN {X 0,Y 347.347,Z 267.644,A -85,B 0,C 180,E1 -15010.249,E2 -15010.249} C_VEL
LIN {X 0,Y 352.203,Z 272.912,A -85,B 0,C 180,E1 -15011.455,E2 -15011.455} C_VEL
LIN {X 0,Y 354.866,Z 275.384,A -85,B 0,C 180,E1 -15012.126,E2 -15012.126} C_VEL
LIN {X 0,Y 359.165,Z 279.61,A -85,B 0,C 180,E1 -15013.306,E2 -15013.306} C_VEL
LIN {X 0,Y 361.917,Z 281.995,A -85,B 0,C 180,E1 -15014.106,E2 -15014.106} C_VEL
LIN {X 0,Y 365.846,Z 285.838,A -85,B 0,C 180,E1 -15015.325,E2 -15015.325} C_VEL
LIN {X 0,Y 369.695,Z 288.971,A -85,B 0,C 180,E1 -15016.615,E2 -15016.615} C_VEL
LIN {X 0,Y 373.669,Z 292.738,A -85,B 0,C 180,E1 -15018.131,E2 -15018.131} C_VEL
LIN {X 0,Y 377.405,Z 295.22,A -85,B 0,C 180,E1 -15019.711,E2 -15019.711} C_VEL
LIN {X 0,Y 378.641,Z 296.156,A -85,B 0,C 180,E1 -15020.316,E2 -15020.316} C_VEL
LIN {X 0,Y 381.246,Z 298.959,A -85,B 0,C 180,E1 -15021.75,E2 -15021.75} C_VEL
LIN {X 0,Y 383.646,Z 300.873,A -85,B 0,C 180,E1 -15023.284,E2 -15023.284} C_VEL
LIN {X 0,Y 385.845,Z 302.139,A -85,B 0,C 180,E1 -15025.046,E2 -15025.046} C_VEL
LIN {X 0,Y 387.489,Z 302.712,A -85,B 0,C 180,E1 -15026.881,E2 -15026.881} C_VEL
LIN {X 0,Y 388.378,Z 303.295,A -85,B 0,C 180,E1 -15028.963,E2 -15028.963} C_VEL
LIN {X 0,Y 388.542,Z 303.227,A -85,B 0,C 180,E1 -15030,E2 -15030} C_VEL
LIN {X 0,Y 388.258,Z 303.182,A -85,B 0,C 180,E1 -15031.556,E2 -15031.556} C_VEL
LIN {X 0,Y 387.234,Z 302.669,A -85,B 0,C 180,E1 -15033.443,E2 -15033.443} C_VEL
LIN {X 0,Y 385.526,Z 301.997,A -85,B 0,C 180,E1 -15035.23,E2 -15035.23} C_VEL
LIN {X 0,Y 383.145,Z 300.518,A -85,B 0,C 180,E1 -15037.072,E2 -15037.072} C_VEL
LIN {X 0,Y 380.459,Z 298.166,A -85,B 0,C 180,E1 -15038.725,E2 -15038.725} C_VEL
LIN {X 0,Y 377.888,Z 295.45,A -85,B 0,C 180,E1 -15040.06,E2 -15040.06} C_VEL
LIN {X 0,Y 374.225,Z 293.2,A -85,B 0,C 180,E1 -15041.637,E2 -15041.637} C_VEL
LIN {X 0,Y 370.283,Z 289.605,A -85,B 0,C 180,E1 -15043.165,E2 -15043.165} C_VEL
LIN {X 0,Y 368.108,Z 287.58,A -85,B 0,C 180,E1 -15043.926,E2 -15043.926} C_VEL
LIN {X 0,Y 363.856,Z 284.083,A -85,B 0,C 180,E1 -15045.298,E2 -15045.298} C_VEL
LIN {X 0,Y 360.454,Z 280.593,A -85,B 0,C 180,E1 -15046.334,E2 -15046.334} C_VEL
LIN {X 0,Y 356.027,Z 276.679,A -85,B 0,C 180,E1 -15047.557,E2 -15047.557} C_VEL
LIN {X 0,Y 353.163,Z 273.705,A -85,B 0,C 180,E1 -15048.309,E2 -15048.309} C_VEL
LIN {X 0,Y 349.166,Z 269.719,A -85,B 0,C 180,E1 -15049.32,E2 -15049.32} C_VEL
LIN {X 0,Y 346.283,Z 266.682,A -85,B 0,C 180,E1 -15049.994,E2 -15049.994} C_VEL
LIN {X 0,Y 342.636,Z 262.414,A -85,B 0,C 180,E1 -15050.86,E2 -15050.86} C_VEL
LIN {X 0,Y 338.649,Z 258.146,A -85,B 0,C 180,E1 -15051.721,E2 -15051.721} C_VEL
LIN {X 0,Y 336.735,Z 255.709,A -85,B 0,C 180,E1 -15052.152,E2 -15052.152} C_VEL
LIN {X 0,Y 333.706,Z 251.945,A -85,B 0,C 180,E1 -15052.774,E2 -15052.774} C_VEL
LIN {X 0,Y 330.474,Z 247.839,A -85,B 0,C 180,E1 -15053.45,E2 -15053.45} C_VEL
LIN {X 0,Y 329.168,Z 245.922,A -85,B 0,C 180,E1 -15053.716,E2 -15053.716} C_VEL
LIN {X 0,Y 327.269,Z 243.479,A -85,B 0,C 180,E1 -15054.08,E2 -15054.08} C_VEL
LIN {X 0,Y 326.717,Z 241.742,A -85,B 0,C 180,E1 -15054.335,E2 -15054.335} C_VEL
LIN {X 0,Y 326.685,Z 241.294,A -85,B 0,C 180,E1 -15054.803,E2 -15054.803} C_VEL
LIN {X 0,Y 326.646,Z 241.281,A -85,B 0,C 180,E1 -15058.251,E2 -15058.251} C_VEL
LIN {X 0,Y 326.586,Z 241.3,A -85,B 0,C 180,E1 -15061.096,E2 -15061.096} C_VEL
LIN {X 0,Y 326.603,Z 241.273,A -85,B 0,C 180,E1 -15064.02,E2 -15064.02} C_VEL
LIN {X 0,Y 326.626,Z 241.298,A -85,B 0,C 180,E1 -15067.239,E2 -15067.239} C_VEL
LIN {X 0,Y 326.599,Z 241.276,A -85,B 0,C 180,E1 -15070.208,E2 -15070.208} C_VEL
LIN {X 0,Y 326.582,Z 241.27,A -85,B 0,C 180,E1 -15073.522,E2 -15073.522} C_VEL
LIN {X 0,Y 326.64,Z 241.296,A -85,B 0,C 180,E1 -15077.016,E2 -15077.016} C_VEL
LIN {X 0,Y 326.642,Z 241.294,A -85,B 0,C 180,E1 -15080.766,E2 -15080.766} C_VEL
LIN {X 0,Y 326.61,Z 241.287,A -85,B 0,C 180,E1 -15084.481,E2 -15084.481} C_VEL
LIN {X 0,Y 326.605,Z 241.296,A -85,B 0,C 180,E1 -15087.456,E2 -15087.456} C_VEL
LIN {X 0,Y 326.658,Z 241.289,A -85,B 0,C 180,E1 -15090.342,E2 -15090.342} C_VEL
LIN {X 0,Y 326.687,Z 241.284,A -85,B 0,C 180,E1 -15094.517,E2 -15094.517} C_VEL
LIN {X 0,Y 326.617,Z 241.292,A -85,B 0,C 180,E1 -15098.544,E2 -15098.544} C_VEL
LIN {X 0,Y 326.743,Z 241.254,A -85,B 0,C 180,E1 -15101.178,E2 -15101.178} C_VEL
LIN {X 0,Y 326.756,Z 241.284,A -85,B 0,C 180,E1 -15105.271,E2 -15105.271} C_VEL
LIN {X 0,Y 326.105,Z 241.367,A -85,B 0,C 180,E1 -15106.3,E2 -15106.3} C_VEL
LIN {X 0,Y 323.239,Z 241.707,A -85,B 0,C 180,E1 -15107.975,E2 -15107.975} C_VEL
LIN {X 0,Y 320.83,Z 241.99,A -85,B 0,C 180,E1 -15109.332,E2 -15109.332} C_VEL
LIN {X 0,Y 319.845,Z 242.109,A -85,B 0,C 180,E1 -15110.382,E2 -15110.382} C_VEL
LIN {X 0,Y 319.791,Z 242.116,A -85,B 0,C 180,E1 -15110.738,E2 -15110.738} C_VEL
LIN {X 0,Y 319.942,Z 242.131,A -85,B 0,C 180,E1 -15113.695,E2 -15113.695} C_VEL
LIN {X 0,Y 319.99,Z 242.109,A -85,B 0,C 180,E1 -15117.483,E2 -15117.483} C_VEL
LIN {X 0,Y 320.13,Z 242.072,A -85,B 0,C 180,E1 -15120.001,E2 -15120.001} C_VEL
LIN {X 0,Y 319.989,Z 242.115,A -85,B 0,C 180,E1 -15122.518,E2 -15122.518} C_VEL
LIN {X 0,Y 319.909,Z 242.131,A -85,B 0,C 180,E1 -15126.307,E2 -15126.307} C_VEL
LIN {X 0,Y 319.735,Z 242.123,A -85,B 0,C 180,E1 -15130.129,E2 -15130.129} C_VEL
LIN {X 0,Y 319.732,Z 242.153,A -85,B 0,C 180,E1 -15133.993,E2 -15133.993} C_VEL
LIN {X 0,Y 319.624,Z 242.142,A -85,B 0,C 180,E1 -15137.93,E2 -15137.93} C_VEL
LIN {X 0,Y 319.597,Z 242.169,A -85,B 0,C 180,E1 -15141.953,E2 -15141.953} C_VEL
LIN {X 0,Y 319.619,Z 242.149,A -85,B 0,C 180,E1 -15146.09,E2 -15146.09} C_VEL
LIN {X 0,Y 319.581,Z 242.168,A -85,B 0,C 180,E1 -15148.935,E2 -15148.935} C_VEL
LIN {X 0,Y 319.531,Z 242.181,A -85,B 0,C 180,E1 -15151.863,E2 -15151.863} C_VEL
LIN {X 0,Y 319.58,Z 242.169,A -85,B 0,C 180,E1 -15155.543,E2 -15155.543} C_VEL
LIN {X 0,Y 319.573,Z 242.178,A -85,B 0,C 180,E1 -15158.009,E2 -15158.009} C_VEL
LIN {X 0,Y 319.527,Z 242.18,A -85,B 0,C 180,E1 -15161.598,E2 -15161.598} C_VEL
LIN {X 0,Y 319.49,Z 242.183,A -85,B 0,C 180,E1 -15165.258,E2 -15165.258} C_VEL
LIN {X 0,Y 319.53,Z 242.16,A -85,B 0,C 180,E1 -15168.712,E2 -15168.712} C_VEL
LIN {X 0,Y 319.579,Z 242.178,A -85,B 0,C 180,E1 -15172.345,E2 -15172.345} C_VEL
LIN {X 0,Y 319.595,Z 242.324,A -85,B 0,C 180,E1 -15176.05,E2 -15176.05} C_VEL
LIN {X 0,Y 320.966,Z 248.803,A -85,B 0,C 180,E1 -15178.646,E2 -15178.646} C_VEL
LIN {X 0,Y 322.404,Z 256.024,A -85,B 0,C 180,E1 -15181.343,E2 -15181.343} C_VEL
LIN {X 0,Y 323.125,Z 260.748,A -85,B 0,C 180,E1 -15183.096,E2 -15183.096} C_VEL
LIN {X 0,Y 322.621,Z 265.849,A -85,B 0,C 180,E1 -15184.827,E2 -15184.827} C_VEL
LIN {X 0,Y 323.525,Z 270.289,A -85,B 0,C 180,E1 -15185.078,E2 -15185.078} C_VEL
LIN {X 0,Y 328.105,Z 292.501,A -85,B 0,C 180,E1 -15185.968,E2 -15185.968} C_VEL
LIN {X 0,Y 330.592,Z 307.258,A -85,B 0,C 180,E1 -15186.501,E2 -15186.501} C_VEL
LIN {X 0,Y 329.207,Z 372.078,A -85,B 0,C 180,E1 -15187.939,E2 -15187.939} C_VEL
LIN {X 0,Y 328.597,Z 382.389,A -85,B 0,C 180,E1 -15188.309,E2 -15188.309} C_VEL
LIN {X 0,Y 327.873,Z 391.903,A -85,B 0,C 180,E1 -15188.794,E2 -15188.794} C_VEL
LIN {X 0,Y 327.011,Z 400.976,A -85,B 0,C 180,E1 -15189.395,E2 -15189.395} C_VEL
LIN {X 0,Y 326.028,Z 410.109,A -85,B 0,C 180,E1 -15190.153,E2 -15190.153} C_VEL
LIN {X 0,Y 324.931,Z 419.104,A -85,B 0,C 180,E1 -15191.069,E2 -15191.069} C_VEL
LIN {X 0,Y 323.701,Z 427.829,A -85,B 0,C 180,E1 -15192.141,E2 -15192.141} C_VEL
LIN {X 0,Y 322.709,Z 435.225,A -85,B 0,C 180,E1 -15193.228,E2 -15193.228} C_VEL
LIN {X 0,Y 321.69,Z 442.649,A -85,B 0,C 180,E1 -15194.518,E2 -15194.518} C_VEL
LIN {X 0,Y 320.844,Z 448.648,A -85,B 0,C 180,E1 -15195.734,E2 -15195.734} C_VEL
LIN {X 0,Y 319.82,Z 455.183,A -85,B 0,C 180,E1 -15197.306,E2 -15197.306} C_VEL
LIN {X 0,Y 319.201,Z 459.686,A -85,B 0,C 180,E1 -15198.571,E2 -15198.571} C_VEL
LIN {X 0,Y 318.539,Z 465.179,A -85,B 0,C 180,E1 -15200.475,E2 -15200.475} C_VEL
LIN {X 0,Y 318.077,Z 469.505,A -85,B 0,C 180,E1 -15202.382,E2 -15202.382} C_VEL
LIN {X 0,Y 317.839,Z 472.776,A -85,B 0,C 180,E1 -15204.291,E2 -15204.291} C_VEL
LIN {X 0,Y 317.786,Z 475.063,A -85,B 0,C 180,E1 -15206.196,E2 -15206.196} C_VEL
LIN {X 0,Y 317.756,Z 476.121,A -85,B 0,C 180,E1 -15207.465,E2 -15207.465} C_VEL
LIN {X 0,Y 317.734,Z 476.71,A -85,B 0,C 180,E1 -15208.733,E2 -15208.733} C_VEL
LIN {X 0,Y 317.734,Z 476.71,A -85,B 0,C 180,E1 -15211.267,E2 -15211.267} C_VEL
LIN {X 0,Y 317.756,Z 476.121,A -85,B 0,C 180,E1 -15212.535,E2 -15212.535} C_VEL
LIN {X 0,Y 317.796,Z 473.673,A -85,B 0,C 180,E1 -15215.075,E2 -15215.075} C_VEL
LIN {X 0,Y 317.985,Z 470.722,A -85,B 0,C 180,E1 -15216.982,E2 -15216.982} C_VEL
LIN {X 0,Y 318.362,Z 466.733,A -85,B 0,C 180,E1 -15218.889,E2 -15218.889} C_VEL
LIN {X 0,Y 318.955,Z 461.602,A -85,B 0,C 180,E1 -15220.795,E2 -15220.795} C_VEL
LIN {X 0,Y 319.63,Z 456.339,A -85,B 0,C 180,E1 -15222.379,E2 -15222.379} C_VEL
LIN {X 0,Y 320.614,Z 450.024,A -85,B 0,C 180,E1 -15223.953,E2 -15223.953} C_VEL
LIN {X 0,Y 321.441,Z 444.071,A -85,B 0,C 180,E1 -15225.211,E2 -15225.211} C_VEL
LIN {X 0,Y 322.41,Z 437.143,A -85,B 0,C 180,E1 -15226.462,E2 -15226.462} C_VEL
LIN {X 0,Y 323.539,Z 428.964,A -85,B 0,C 180,E1 -15227.705,E2 -15227.705} C_VEL
LIN {X 0,Y 324.74,Z 420.455,A -85,B 0,C 180,E1 -15228.779,E2 -15228.779} C_VEL
LIN {X 0,Y 325.857,Z 411.741,A -85,B 0,C 180,E1 -15229.694,E2 -15229.694} C_VEL
LIN {X 0,Y 326.906,Z 401.983,A -85,B 0,C 180,E1 -15230.53,E2 -15230.53} C_VEL
LIN {X 0,Y 327.915,Z 391.904,A -85,B 0,C 180,E1 -15231.203,E2 -15231.203} C_VEL
LIN {X 0,Y 328.624,Z 382.39,A -85,B 0,C 180,E1 -15231.69,E2 -15231.69} C_VEL
LIN {X 0,Y 329.181,Z 372.077,A -85,B 0,C 180,E1 -15232.063,E2 -15232.063} C_VEL
LIN {X 0,Y 330.529,Z 306.739,A -85,B 0,C 180,E1 -15233.516,E2 -15233.516} C_VEL
LIN {X 0,Y 326.36,Z 283.312,A -85,B 0,C 180,E1 -15234.384,E2 -15234.384} C_VEL
LIN {X 0,Y 322.632,Z 266.163,A -85,B 0,C 180,E1 -15235.127,E2 -15235.127} C_VEL
LIN {X 0,Y 322.728,Z 264.689,A -85,B 0,C 180,E1 -15235.508,E2 -15235.508} C_VEL
LIN {X 0,Y 323.105,Z 260.772,A -85,B 0,C 180,E1 -15236.897,E2 -15236.897} C_VEL
LIN {X 0,Y 321.934,Z 253.528,A -85,B 0,C 180,E1 -15239.605,E2 -15239.605} C_VEL
LIN {X 0,Y 320.174,Z 244.931,A -85,B 0,C 180,E1 -15242.907,E2 -15242.907} C_VEL
LIN {X 0,Y 319.613,Z 242.258,A -85,B 0,C 180,E1 -15244.01,E2 -15244.01} C_VEL
LIN {X 0,Y 319.575,Z 242.178,A -85,B 0,C 180,E1 -15248.008,E2 -15248.008} C_VEL
LIN {X 0,Y 319.527,Z 242.163,A -85,B 0,C 180,E1 -15251.596,E2 -15251.596} C_VEL
LIN {X 0,Y 319.49,Z 242.18,A -85,B 0,C 180,E1 -15255.257,E2 -15255.257} C_VEL
LIN {X 0,Y 319.53,Z 242.179,A -85,B 0,C 180,E1 -15258.711,E2 -15258.711} C_VEL
LIN {X 0,Y 319.562,Z 242.178,A -85,B 0,C 180,E1 -15262.348,E2 -15262.348} C_VEL
LIN {X 0,Y 319.559,Z 242.162,A -85,B 0,C 180,E1 -15265.123,E2 -15265.123} C_VEL
LIN {X 0,Y 319.567,Z 242.178,A -85,B 0,C 180,E1 -15269.059,E2 -15269.059} C_VEL
LIN {X 0,Y 319.606,Z 242.15,A -85,B 0,C 180,E1 -15272.497,E2 -15272.497} C_VEL
LIN {X 0,Y 319.604,Z 242.163,A -85,B 0,C 180,E1 -15275.303,E2 -15275.303} C_VEL
LIN {X 0,Y 319.597,Z 242.169,A -85,B 0,C 180,E1 -15278.047,E2 -15278.047} C_VEL
LIN {X 0,Y 319.624,Z 242.142,A -85,B 0,C 180,E1 -15282.07,E2 -15282.07} C_VEL
LIN {X 0,Y 319.732,Z 242.153,A -85,B 0,C 180,E1 -15286.007,E2 -15286.007} C_VEL
LIN {X 0,Y 319.735,Z 242.123,A -85,B 0,C 180,E1 -15289.871,E2 -15289.871} C_VEL
LIN {X 0,Y 319.909,Z 242.131,A -85,B 0,C 180,E1 -15293.693,E2 -15293.693} C_VEL
LIN {X 0,Y 319.989,Z 242.115,A -85,B 0,C 180,E1 -15297.482,E2 -15297.482} C_VEL
LIN {X 0,Y 320.13,Z 242.072,A -85,B 0,C 180,E1 -15299.999,E2 -15299.999} C_VEL
LIN {X 0,Y 319.99,Z 242.109,A -85,B 0,C 180,E1 -15302.517,E2 -15302.517} C_VEL
LIN {X 0,Y 319.922,Z 242.129,A -85,B 0,C 180,E1 -15306.574,E2 -15306.574} C_VEL
LIN {X 0,Y 319.751,Z 242.12,A -85,B 0,C 180,E1 -15310.127,E2 -15310.127} C_VEL
LIN {X 0,Y 319.729,Z 242.159,A -85,B 0,C 180,E1 -15314.724,E2 -15314.724} C_VEL
LIN {X 0,Y 319.687,Z 242.132,A -85,B 0,C 180,E1 -15319.037,E2 -15319.037} C_VEL
LIN {X 0,Y 319.558,Z 242.178,A -85,B 0,C 180,E1 -15323.32,E2 -15323.32} C_VEL
LIN {X 0,Y 319.616,Z 242.153,A -85,B 0,C 180,E1 -15326.089,E2 -15326.089} C_VEL
LIN {X 0,Y 319.587,Z 242.164,A -85,B 0,C 180,E1 -15328.933,E2 -15328.933} C_VEL
LIN {X 0,Y 319.529,Z 242.185,A -85,B 0,C 180,E1 -15331.861,E2 -15331.861} C_VEL
LIN {X 0,Y 319.577,Z 242.163,A -85,B 0,C 180,E1 -15335.542,E2 -15335.542} C_VEL
LIN {X 0,Y 319.595,Z 242.178,A -85,B 0,C 180,E1 -15338.004,E2 -15338.004} C_VEL
LIN {X 0,Y 319.598,Z 242.162,A -85,B 0,C 180,E1 -15341.612,E2 -15341.612} C_VEL
LIN {X 0,Y 319.584,Z 242.17,A -85,B 0,C 180,E1 -15344.725,E2 -15344.725} C_VEL
LIN {X 0,Y 319.53,Z 242.137,A -85,B 0,C 180,E1 -15348.712,E2 -15348.712} C_VEL
LIN {X 0,Y 319.578,Z 242.177,A -85,B 0,C 180,E1 -15352.343,E2 -15352.343} C_VEL
LIN {X 0,Y 319.556,Z 242.148,A -85,B 0,C 180,E1 -15355.123,E2 -15355.123} C_VEL
LIN {X 0,Y 319.562,Z 242.172,A -85,B 0,C 180,E1 -15359.059,E2 -15359.059} C_VEL
LIN {X 0,Y 319.602,Z 242.171,A -85,B 0,C 180,E1 -15362.498,E2 -15362.498} C_VEL
LIN {X 0,Y 319.676,Z 242.391,A -85,B 0,C 180,E1 -15364.614,E2 -15364.614} C_VEL
LIN {X 0,Y 319.92,Z 243.459,A -85,B 0,C 180,E1 -15364.853,E2 -15364.853} C_VEL
LIN {X 0,Y 321.68,Z 246.339,A -85,B 0,C 180,E1 -15365.191,E2 -15365.191} C_VEL
LIN {X 0,Y 324.766,Z 250.848,A -85,B 0,C 180,E1 -15365.751,E2 -15365.751} C_VEL
LIN {X 0,Y 326.716,Z 253.439,A -85,B 0,C 180,E1 -15366.125,E2 -15366.125} C_VEL
LIN {X 0,Y 330.78,Z 258.549,A -85,B 0,C 180,E1 -15366.921,E2 -15366.921} C_VEL
LIN {X 0,Y 336.02,Z 264.755,A -85,B 0,C 180,E1 -15367.994,E2 -15367.994} C_VEL
LIN {X 0,Y 340.983,Z 270.245,A -85,B 0,C 180,E1 -15369.076,E2 -15369.076} C_VEL
LIN {X 0,Y 346.362,Z 275.83,A -85,B 0,C 180,E1 -15370.311,E2 -15370.311} C_VEL
LIN {X 0,Y 350.372,Z 279.778,A -85,B 0,C 180,E1 -15371.28,E2 -15371.28} C_VEL
LIN {X 0,Y 355.887,Z 285.172,A -85,B 0,C 180,E1 -15372.713,E2 -15372.713} C_VEL
LIN {X 0,Y 359.776,Z 288.466,A -85,B 0,C 180,E1 -15373.784,E2 -15373.784} C_VEL
LIN {X 0,Y 364.001,Z 292.516,A -85,B 0,C 180,E1 -15375.073,E2 -15375.073} C_VEL
LIN {X 0,Y 367.974,Z 295.697,A -85,B 0,C 180,E1 -15376.368,E2 -15376.368} C_VEL
LIN {X 0,Y 372.207,Z 299.581,A -85,B 0,C 180,E1 -15377.937,E2 -15377.937} C_VEL
LIN {X 0,Y 376.1,Z 302.113,A -85,B 0,C 180,E1 -15379.54,E2 -15379.54} C_VEL
LIN {X 0,Y 377.407,Z 303.141,A -85,B 0,C 180,E1 -15380.169,E2 -15380.169} C_VEL
LIN {X 0,Y 380.162,Z 305.986,A -85,B 0,C 180,E1 -15381.649,E2 -15381.649} C_VEL
LIN {X 0,Y 382.58,Z 307.842,A -85,B 0,C 180,E1 -15383.16,E2 -15383.16} C_VEL
LIN {X 0,Y 384.637,Z 309.028,A -85,B 0,C 180,E1 -15384.758,E2 -15384.758} C_VEL
LIN {X 0,Y 386.062,Z 309.613,A -85,B 0,C 180,E1 -15386.193,E2 -15386.193} C_VEL
LIN {X 0,Y 387.299,Z 310.162,A -85,B 0,C 180,E1 -15388.18,E2 -15388.18} C_VEL
LIN {X 0,Y 387.677,Z 310.274,A -85,B 0,C 180,E1 -15390,E2 -15390} C_VEL
LIN {X 0,Y 387.389,Z 310.23,A -85,B 0,C 180,E1 -15391.559,E2 -15391.559} C_VEL
LIN {X 0,Y 386.606,Z 309.789,A -85,B 0,C 180,E1 -15393.126,E2 -15393.126} C_VEL
LIN {X 0,Y 384.954,Z 309.191,A -85,B 0,C 180,E1 -15394.966,E2 -15394.966} C_VEL
LIN {X 0,Y 382.579,Z 307.847,A -85,B 0,C 180,E1 -15396.84,E2 -15396.84} C_VEL
LIN {X 0,Y 379.898,Z 305.708,A -85,B 0,C 180,E1 -15398.511,E2 -15398.511} C_VEL
LIN {X 0,Y 376.433,Z 302.253,A -85,B 0,C 180,E1 -15400.316,E2 -15400.316} C_VEL
LIN {X 0,Y 372.429,Z 299.736,A -85,B 0,C 180,E1 -15401.98,E2 -15401.98} C_VEL
LIN {X 0,Y 368.346,Z 296.068,A -85,B 0,C 180,E1 -15403.506,E2 -15403.506} C_VEL
LIN {X 0,Y 366.154,Z 294.122,A -85,B 0,C 180,E1 -15404.239,E2 -15404.239} C_VEL
LIN {X 0,Y 361.515,Z 290.352,A -85,B 0,C 180,E1 -15405.684,E2 -15405.684} C_VEL
LIN {X 0,Y 358.078,Z 286.93,A -85,B 0,C 180,E1 -15406.696,E2 -15406.696} C_VEL
LIN {X 0,Y 353.448,Z 282.85,A -85,B 0,C 180,E1 -15407.942,E2 -15407.942} C_VEL
LIN {X 0,Y 350.586,Z 279.953,A -85,B 0,C 180,E1 -15408.666,E2 -15408.666} C_VEL
LIN {X 0,Y 346.501,Z 276.03,A -85,B 0,C 180,E1 -15409.655,E2 -15409.655} C_VEL
LIN {X 0,Y 343.245,Z 272.581,A -85,B 0,C 180,E1 -15410.423,E2 -15410.423} C_VEL
LIN {X 0,Y 335.24,Z 263.807,A -85,B 0,C 180,E1 -15412.17,E2 -15412.17} C_VEL
LIN {X 0,Y 331.945,Z 259.982,A -85,B 0,C 180,E1 -15412.837,E2 -15412.837} C_VEL
LIN {X 0,Y 328.505,Z 255.671,A -85,B 0,C 180,E1 -15413.535,E2 -15413.535} C_VEL
LIN {X 0,Y 324.51,Z 250.538,A -85,B 0,C 180,E1 -15414.298,E2 -15414.298} C_VEL
LIN {X 0,Y 321.314,Z 245.932,A -85,B 0,C 180,E1 -15414.871,E2 -15414.871} C_VEL
LIN {X 0,Y 319.834,Z 243.073,A -85,B 0,C 180,E1 -15415.196,E2 -15415.196} C_VEL
LIN {X 0,Y 319.659,Z 242.224,A -85,B 0,C 180,E1 -15415.517,E2 -15415.517} C_VEL
LIN {X 0,Y 319.576,Z 242.155,A -85,B 0,C 180,E1 -15418.935,E2 -15418.935} C_VEL
LIN {X 0,Y 319.527,Z 242.186,A -85,B 0,C 180,E1 -15421.862,E2 -15421.862} C_VEL
LIN {X 0,Y 319.576,Z 242.15,A -85,B 0,C 180,E1 -15425.543,E2 -15425.543} C_VEL
LIN {X 0,Y 319.594,Z 242.178,A -85,B 0,C 180,E1 -15428.005,E2 -15428.005} C_VEL
LIN {X 0,Y 319.527,Z 242.135,A -85,B 0,C 180,E1 -15431.598,E2 -15431.598} C_VEL
LIN {X 0,Y 319.584,Z 242.17,A -85,B 0,C 180,E1 -15435.275,E2 -15435.275} C_VEL
LIN {X 0,Y 319.58,Z 242.163,A -85,B 0,C 180,E1 -15438.721,E2 -15438.721} C_VEL
LIN {X 0,Y 319.595,Z 242.176,A -85,B 0,C 180,E1 -15442.34,E2 -15442.34} C_VEL
LIN {X 0,Y 319.557,Z 242.161,A -85,B 0,C 180,E1 -15445.124,E2 -15445.124} C_VEL
LIN {X 0,Y 319.567,Z 242.178,A -85,B 0,C 180,E1 -15449.059,E2 -15449.059} C_VEL
LIN {X 0,Y 319.605,Z 242.146,A -85,B 0,C 180,E1 -15452.499,E2 -15452.499} C_VEL
LIN {X 0,Y 319.6,Z 242.169,A -85,B 0,C 180,E1 -15455.304,E2 -15455.304} C_VEL
LIN {X 0,Y 319.6,Z 242.153,A -85,B 0,C 180,E1 -15459.401,E2 -15459.401} C_VEL
LIN {X 0,Y 319.656,Z 242.144,A -85,B 0,C 180,E1 -15462.074,E2 -15462.074} C_VEL
LIN {X 0,Y 319.731,Z 242.156,A -85,B 0,C 180,E1 -15466.008,E2 -15466.008} C_VEL
LIN {X 0,Y 319.751,Z 242.12,A -85,B 0,C 180,E1 -15469.873,E2 -15469.873} C_VEL
LIN {X 0,Y 319.791,Z 242.116,A -85,B 0,C 180,E1 -15470.738,E2 -15470.738} C_VEL
LIN {X 0,Y 319.514,Z 242.16,A -85,B 0,C 180,E1 -15471.442,E2 -15471.442} C_VEL
LIN {X 0,Y 317.543,Z 242.421,A -85,B 0,C 180,E1 -15472.82,E2 -15472.82} C_VEL
LIN {X 0,Y 313.744,Z 242.906,A -85,B 0,C 180,E1 -15474.885,E2 -15474.885} C_VEL
LIN {X 0,Y 312.755,Z 243.023,A -85,B 0,C 180,E1 -15475.96,E2 -15475.96} C_VEL
LIN {X 0,Y 312.718,Z 243.024,A -85,B 0,C 180,E1 -15476.324,E2 -15476.324} C_VEL
LIN {X 0,Y 312.988,Z 242.967,A -85,B 0,C 180,E1 -15478.714,E2 -15478.714} C_VEL
LIN {X 0,Y 312.988,Z 242.971,A -85,B 0,C 180,E1 -15481.287,E2 -15481.287} C_VEL
LIN {X 0,Y 312.707,Z 243.033,A -85,B 0,C 180,E1 -15485.158,E2 -15485.158} C_VEL
LIN {X 0,Y 312.817,Z 243,A -85,B 0,C 180,E1 -15487.748,E2 -15487.748} C_VEL
LIN {X 0,Y 312.663,Z 243.021,A -85,B 0,C 180,E1 -15491.672,E2 -15491.672} C_VEL
LIN {X 0,Y 312.668,Z 243.035,A -85,B 0,C 180,E1 -15494.866,E2 -15494.866} C_VEL
LIN {X 0,Y 312.592,Z 243.016,A -85,B 0,C 180,E1 -15499.217,E2 -15499.217} C_VEL
LIN {X 0,Y 312.546,Z 243.053,A -85,B 0,C 180,E1 -15502.79,E2 -15502.79} C_VEL
LIN {X 0,Y 312.597,Z 243.025,A -85,B 0,C 180,E1 -15505.934,E2 -15505.934} C_VEL
LIN {X 0,Y 312.539,Z 243.05,A -85,B 0,C 180,E1 -15509.651,E2 -15509.651} C_VEL
LIN {X 0,Y 312.52,Z 243.036,A -85,B 0,C 180,E1 -15513.689,E2 -15513.689} C_VEL
LIN {X 0,Y 312.526,Z 243.055,A -85,B 0,C 180,E1 -15517.386,E2 -15517.386} C_VEL
LIN {X 0,Y 312.491,Z 243.049,A -85,B 0,C 180,E1 -15520.71,E2 -15520.71} C_VEL
LIN {X 0,Y 312.453,Z 243.056,A -85,B 0,C 180,E1 -15524.21,E2 -15524.21} C_VEL
LIN {X 0,Y 312.486,Z 243.047,A -85,B 0,C 180,E1 -15527.919,E2 -15527.919} C_VEL
LIN {X 0,Y 312.537,Z 243.054,A -85,B 0,C 180,E1 -15531.911,E2 -15531.911} C_VEL
LIN {X 0,Y 312.56,Z 243.224,A -85,B 0,C 180,E1 -15535.602,E2 -15535.602} C_VEL
LIN {X 0,Y 314.049,Z 250.292,A -85,B 0,C 180,E1 -15538.478,E2 -15538.478} C_VEL
LIN {X 0,Y 315.524,Z 257.796,A -85,B 0,C 180,E1 -15541.387,E2 -15541.387} C_VEL
LIN {X 0,Y 316.15,Z 262.548,A -85,B 0,C 180,E1 -15543.195,E2 -15543.195} C_VEL
LIN {X 0,Y 315.866,Z 265.676,A -85,B 0,C 180,E1 -15544.255,E2 -15544.255} C_VEL
LIN {X 0,Y 316.791,Z 270.129,A -85,B 0,C 180,E1 -15544.512,E2 -15544.512} C_VEL
LIN {X 0,Y 321.757,Z 294.357,A -85,B 0,C 180,E1 -15545.512,E2 -15545.512} C_VEL
LIN {X 0,Y 324.103,Z 308.832,A -85,B 0,C 180,E1 -15546.043,E2 -15546.043} C_VEL
LIN {X 0,Y 322.623,Z 371.885,A -85,B 0,C 180,E1 -15547.464,E2 -15547.464} C_VEL
LIN {X 0,Y 322.008,Z 382.196,A -85,B 0,C 180,E1 -15547.841,E2 -15547.841} C_VEL
LIN {X 0,Y 321.27,Z 391.71,A -85,B 0,C 180,E1 -15548.337,E2 -15548.337} C_VEL
LIN {X 0,Y 320.261,Z 401.79,A -85,B 0,C 180,E1 -15549.024,E2 -15549.024} C_VEL
LIN {X 0,Y 319.176,Z 411.548,A -85,B 0,C 180,E1 -15549.876,E2 -15549.876} C_VEL
LIN {X 0,Y 317.842,Z 421.613,A -85,B 0,C 180,E1 -15550.965,E2 -15550.965} C_VEL
LIN {X 0,Y 316.17,Z 433.112,A -85,B 0,C 180,E1 -15552.537,E2 -15552.537} C_VEL
LIN {X 0,Y 315.031,Z 441.381,A -85,B 0,C 180,E1 -15553.962,E2 -15553.962} C_VEL
LIN {X 0,Y 313.94,Z 448.455,A -85,B 0,C 180,E1 -15555.413,E2 -15555.413} C_VEL
LIN {X 0,Y 312.886,Z 454.99,A -85,B 0,C 180,E1 -15557.02,E2 -15557.02} C_VEL
LIN {X 0,Y 312.195,Z 459.492,A -85,B 0,C 180,E1 -15558.311,E2 -15558.311} C_VEL
LIN {X 0,Y 311.493,Z 464.985,A -85,B 0,C 180,E1 -15560.258,E2 -15560.258} C_VEL
LIN {X 0,Y 311.02,Z 469.311,A -85,B 0,C 180,E1 -15562.208,E2 -15562.208} C_VEL
LIN {X 0,Y 310.826,Z 471.68,A -85,B 0,C 180,E1 -15563.509,E2 -15563.509} C_VEL
LIN {X 0,Y 310.706,Z 473.48,A -85,B 0,C 180,E1 -15564.809,E2 -15564.809} C_VEL
LIN {X 0,Y 310.679,Z 475.929,A -85,B 0,C 180,E1 -15567.407,E2 -15567.407} C_VEL
LIN {X 0,Y 310.649,Z 476.518,A -85,B 0,C 180,E1 -15568.704,E2 -15568.704} C_VEL
LIN {X 0,Y 310.649,Z 476.518,A -85,B 0,C 180,E1 -15571.296,E2 -15571.296} C_VEL
LIN {X 0,Y 310.679,Z 475.929,A -85,B 0,C 180,E1 -15572.593,E2 -15572.593} C_VEL
LIN {X 0,Y 310.7,Z 473.48,A -85,B 0,C 180,E1 -15575.191,E2 -15575.191} C_VEL
LIN {X 0,Y 310.919,Z 470.529,A -85,B 0,C 180,E1 -15577.142,E2 -15577.142} C_VEL
LIN {X 0,Y 311.308,Z 466.539,A -85,B 0,C 180,E1 -15579.093,E2 -15579.093} C_VEL
LIN {X 0,Y 311.954,Z 461.409,A -85,B 0,C 180,E1 -15581.04,E2 -15581.04} C_VEL
LIN {X 0,Y 312.669,Z 456.145,A -85,B 0,C 180,E1 -15582.659,E2 -15582.659} C_VEL
LIN {X 0,Y 313.687,Z 449.83,A -85,B 0,C 180,E1 -15584.267,E2 -15584.267} C_VEL
LIN {X 0,Y 314.798,Z 442.682,A -85,B 0,C 180,E1 -15585.784,E2 -15585.784} C_VEL
LIN {X 0,Y 315.886,Z 435.031,A -85,B 0,C 180,E1 -15587.145,E2 -15587.145} C_VEL
LIN {X 0,Y 317.102,Z 426.502,A -85,B 0,C 180,E1 -15588.411,E2 -15588.411} C_VEL
LIN {X 0,Y 318.603,Z 416.209,A -85,B 0,C 180,E1 -15589.657,E2 -15589.657} C_VEL
LIN {X 0,Y 320.05,Z 403.804,A -85,B 0,C 180,E1 -15590.822,E2 -15590.822} C_VEL
LIN {X 0,Y 321.195,Z 392.999,A -85,B 0,C 180,E1 -15591.584,E2 -15591.584} C_VEL
LIN {X 0,Y 321.972,Z 383.071,A -85,B 0,C 180,E1 -15592.119,E2 -15592.119} C_VEL
LIN {X 0,Y 322.575,Z 373.217,A -85,B 0,C 180,E1 -15592.497,E2 -15592.497} C_VEL
LIN {X 0,Y 323.23,Z 347.743,A -85,B 0,C 180,E1 -15593.103,E2 -15593.103} C_VEL
LIN {X 0,Y 323.938,Z 307.02,A -85,B 0,C 180,E1 -15594.013,E2 -15594.013} C_VEL
LIN {X 0,Y 319.817,Z 284.038,A -85,B 0,C 180,E1 -15594.895,E2 -15594.895} C_VEL
LIN {X 0,Y 315.857,Z 266.017,A -85,B 0,C 180,E1 -15595.7,E2 -15595.7} C_VEL
LIN {X 0,Y 315.96,Z 264.588,A -85,B 0,C 180,E1 -15596.06,E2 -15596.06} C_VEL
LIN {X 0,Y 316.121,Z 261.445,A -85,B 0,C 180,E1 -15597.216,E2 -15597.216} C_VEL
LIN {X 0,Y 314.763,Z 253.831,A -85,B 0,C 180,E1 -15600.157,E2 -15600.157} C_VEL
LIN {X 0,Y 313.202,Z 246.237,A -85,B 0,C 180,E1 -15603.161,E2 -15603.161} C_VEL
LIN {X 0,Y 312.53,Z 243.101,A -85,B 0,C 180,E1 -15604.5,E2 -15604.5} C_VEL
LIN {X 0,Y 312.537,Z 243.054,A -85,B 0,C 180,E1 -15608.089,E2 -15608.089} C_VEL
LIN {X 0,Y 312.486,Z 243.046,A -85,B 0,C 180,E1 -15612.081,E2 -15612.081} C_VEL
LIN {X 0,Y 312.46,Z 243.057,A -85,B 0,C 180,E1 -15616.034,E2 -15616.034} C_VEL
LIN {X 0,Y 312.506,Z 243.044,A -85,B 0,C 180,E1 -15619.874,E2 -15619.874} C_VEL
LIN {X 0,Y 312.526,Z 243.055,A -85,B 0,C 180,E1 -15622.614,E2 -15622.614} C_VEL
LIN {X 0,Y 312.52,Z 243.036,A -85,B 0,C 180,E1 -15626.311,E2 -15626.311} C_VEL
LIN {X 0,Y 312.539,Z 243.05,A -85,B 0,C 180,E1 -15630.349,E2 -15630.349} C_VEL
LIN {X 0,Y 312.597,Z 243.025,A -85,B 0,C 180,E1 -15634.066,E2 -15634.066} C_VEL
LIN {X 0,Y 312.588,Z 243.045,A -85,B 0,C 180,E1 -15637.528,E2 -15637.528} C_VEL
LIN {X 0,Y 312.589,Z 243.015,A -85,B 0,C 180,E1 -15641.653,E2 -15641.653} C_VEL
LIN {X 0,Y 312.686,Z 243.032,A -85,B 0,C 180,E1 -15645.685,E2 -15645.685} C_VEL
LIN {X 0,Y 312.685,Z 243.002,A -85,B 0,C 180,E1 -15649.641,E2 -15649.641} C_VEL
LIN {X 0,Y 312.817,Z 243,A -85,B 0,C 180,E1 -15652.252,E2 -15652.252} C_VEL
LIN {X 0,Y 312.707,Z 243.033,A -85,B 0,C 180,E1 -15654.842,E2 -15654.842} C_VEL
LIN {X 0,Y 312.988,Z 242.971,A -85,B 0,C 180,E1 -15658.713,E2 -15658.713} C_VEL
LIN {X 0,Y 312.988,Z 242.967,A -85,B 0,C 180,E1 -15661.286,E2 -15661.286} C_VEL
LIN {X 0,Y 312.714,Z 243.031,A -85,B 0,C 180,E1 -15665.157,E2 -15665.157} C_VEL
LIN {X 0,Y 312.852,Z 243.001,A -85,B 0,C 180,E1 -15667.745,E2 -15667.745} C_VEL
LIN {X 0,Y 312.668,Z 243.019,A -85,B 0,C 180,E1 -15671.671,E2 -15671.671} C_VEL
LIN {X 0,Y 312.698,Z 243.033,A -85,B 0,C 180,E1 -15674.887,E2 -15674.887} C_VEL
LIN {X 0,Y 312.607,Z 243.013,A -85,B 0,C 180,E1 -15679.224,E2 -15679.224} C_VEL
LIN {X 0,Y 312.524,Z 243.056,A -85,B 0,C 180,E1 -15682.78,E2 -15682.78} C_VEL
LIN {X 0,Y 312.594,Z 243.029,A -85,B 0,C 180,E1 -15685.933,E2 -15685.933} C_VEL
LIN {X 0,Y 312.542,Z 243.047,A -85,B 0,C 180,E1 -15689.649,E2 -15689.649} C_VEL
LIN {X 0,Y 312.516,Z 243.041,A -85,B 0,C 180,E1 -15693.688,E2 -15693.688} C_VEL
LIN {X 0,Y 312.548,Z 243.053,A -85,B 0,C 180,E1 -15697.381,E2 -15697.381} C_VEL
LIN {X 0,Y 312.524,Z 243.039,A -85,B 0,C 180,E1 -15700.703,E2 -15700.703} C_VEL
LIN {X 0,Y 312.539,Z 243.05,A -85,B 0,C 180,E1 -15704.193,E2 -15704.193} C_VEL
LIN {X 0,Y 312.486,Z 243.01,A -85,B 0,C 180,E1 -15707.917,E2 -15707.917} C_VEL
LIN {X 0,Y 312.553,Z 243.056,A -85,B 0,C 180,E1 -15711.905,E2 -15711.905} C_VEL
LIN {X 0,Y 312.502,Z 243.027,A -85,B 0,C 180,E1 -15715.79,E2 -15715.79} C_VEL
LIN {X 0,Y 312.517,Z 243.053,A -85,B 0,C 180,E1 -15718.853,E2 -15718.853} C_VEL
LIN {X 0,Y 312.566,Z 243.035,A -85,B 0,C 180,E1 -15721.824,E2 -15721.824} C_VEL
LIN {X 0,Y 312.603,Z 243.217,A -85,B 0,C 180,E1 -15723.741,E2 -15723.741} C_VEL
LIN {X 0,Y 312.824,Z 244.105,A -85,B 0,C 180,E1 -15723.98,E2 -15723.98} C_VEL
LIN {X 0,Y 314.289,Z 246.825,A -85,B 0,C 180,E1 -15724.259,E2 -15724.259} C_VEL
LIN {X 0,Y 317.383,Z 251.455,A -85,B 0,C 180,E1 -15724.753,E2 -15724.753} C_VEL
LIN {X 0,Y 320.824,Z 256.319,A -85,B 0,C 180,E1 -15725.351,E2 -15725.351} C_VEL
LIN {X 0,Y 325.313,Z 261.814,A -85,B 0,C 180,E1 -15726.151,E2 -15726.151} C_VEL
LIN {X 0,Y 330.102,Z 267.429,A -85,B 0,C 180,E1 -15727.068,E2 -15727.068} C_VEL
LIN {X 0,Y 334.796,Z 272.782,A -85,B 0,C 180,E1 -15728.021,E2 -15728.021} C_VEL
LIN {X 0,Y 340.968,Z 279.245,A -85,B 0,C 180,E1 -15729.347,E2 -15729.347} C_VEL
LIN {X 0,Y 347.399,Z 285.739,A -85,B 0,C 180,E1 -15730.834,E2 -15730.834} C_VEL
LIN {X 0,Y 351.028,Z 289.238,A -85,B 0,C 180,E1 -15731.742,E2 -15731.742} C_VEL
LIN {X 0,Y 355.517,Z 293.117,A -85,B 0,C 180,E1 -15732.906,E2 -15732.906} C_VEL
LIN {X 0,Y 361.31,Z 298.536,A -85,B 0,C 180,E1 -15734.572,E2 -15734.572} C_VEL
LIN {X 0,Y 366.018,Z 302.195,A -85,B 0,C 180,E1 -15736.053,E2 -15736.053} C_VEL
LIN {X 0,Y 370.012,Z 305.857,A -85,B 0,C 180,E1 -15737.482,E2 -15737.482} C_VEL
LIN {X 0,Y 373.581,Z 308.355,A -85,B 0,C 180,E1 -15738.882,E2 -15738.882} C_VEL
LIN {X 0,Y 375.881,Z 309.798,A -85,B 0,C 180,E1 -15739.873,E2 -15739.873} C_VEL
LIN {X 0,Y 378.947,Z 312.876,A -85,B 0,C 180,E1 -15741.468,E2 -15741.468} C_VEL
LIN {X 0,Y 381.669,Z 314.907,A -85,B 0,C 180,E1 -15743.143,E2 -15743.143} C_VEL
LIN {X 0,Y 384.063,Z 316.239,A -85,B 0,C 180,E1 -15745.023,E2 -15745.023} C_VEL
LIN {X 0,Y 385.734,Z 316.806,A -85,B 0,C 180,E1 -15746.867,E2 -15746.867} C_VEL
LIN {X 0,Y 386.655,Z 317.383,A -85,B 0,C 180,E1 -15748.959,E2 -15748.959} C_VEL
LIN {X 0,Y 386.812,Z 317.32,A -85,B 0,C 180,E1 -15750,E2 -15750} C_VEL
LIN {X 0,Y 386.523,Z 317.255,A -85,B 0,C 180,E1 -15751.563,E2 -15751.563} C_VEL
LIN {X 0,Y 385.729,Z 316.835,A -85,B 0,C 180,E1 -15753.133,E2 -15753.133} C_VEL
LIN {X 0,Y 384.063,Z 316.241,A -85,B 0,C 180,E1 -15754.977,E2 -15754.977} C_VEL
LIN {X 0,Y 381.668,Z 314.912,A -85,B 0,C 180,E1 -15756.856,E2 -15756.856} C_VEL
LIN {X 0,Y 378.694,Z 312.643,A -85,B 0,C 180,E1 -15758.683,E2 -15758.683} C_VEL
LIN {X 0,Y 375.156,Z 309.177,A -85,B 0,C 180,E1 -15760.465,E2 -15760.465} C_VEL
LIN {X 0,Y 371.149,Z 306.69,A -85,B 0,C 180,E1 -15762.097,E2 -15762.097} C_VEL
LIN {X 0,Y 367.011,Z 303.188,A -85,B 0,C 180,E1 -15763.611,E2 -15763.611} C_VEL
LIN {X 0,Y 364.071,Z 300.572,A -85,B 0,C 180,E1 -15764.592,E2 -15764.592} C_VEL
LIN {X 0,Y 359.247,Z 296.65,A -85,B 0,C 180,E1 -15766.049,E2 -15766.049} C_VEL
LIN {X 0,Y 355.5,Z 293.111,A -85,B 0,C 180,E1 -15767.098,E2 -15767.098} C_VEL
LIN {X 0,Y 351.022,Z 289.255,A -85,B 0,C 180,E1 -15768.259,E2 -15768.259} C_VEL
LIN {X 0,Y 347.251,Z 285.565,A -85,B 0,C 180,E1 -15769.203,E2 -15769.203} C_VEL
LIN {X 0,Y 342.661,Z 280.965,A -85,B 0,C 180,E1 -15770.272,E2 -15770.272} C_VEL
LIN {X 0,Y 336.602,Z 274.695,A -85,B 0,C 180,E1 -15771.594,E2 -15771.594} C_VEL
LIN {X 0,Y 331.269,Z 268.89,A -85,B 0,C 180,E1 -15772.69,E2 -15772.69} C_VEL
LIN {X 0,Y 325.992,Z 262.605,A -85,B 0,C 180,E1 -15773.722,E2 -15773.722} C_VEL
LIN {X 0,Y 322.171,Z 257.941,A -85,B 0,C 180,E1 -15774.423,E2 -15774.423} C_VEL
LIN {X 0,Y 318.202,Z 252.751,A -85,B 0,C 180,E1 -15775.104,E2 -15775.104} C_VEL
LIN {X 0,Y 314.994,Z 247.911,A -85,B 0,C 180,E1 -15775.629,E2 -15775.629} C_VEL
LIN {X 0,Y 312.909,Z 244.39,A -85,B 0,C 180,E1 -15775.986,E2 -15775.986} C_VEL
LIN {X 0,Y 312.617,Z 243.334,A -85,B 0,C 180,E1 -15776.194,E2 -15776.194} C_VEL
LIN {X 0,Y 312.549,Z 243.054,A -85,B 0,C 180,E1 -15776.726,E2 -15776.726} C_VEL
LIN {X 0,Y 312.534,Z 243.031,A -85,B 0,C 180,E1 -15779.651,E2 -15779.651} C_VEL
LIN {X 0,Y 312.515,Z 243.03,A -85,B 0,C 180,E1 -15783.689,E2 -15783.689} C_VEL
LIN {X 0,Y 312.537,Z 243.054,A -85,B 0,C 180,E1 -15787.383,E2 -15787.383} C_VEL
LIN {X 0,Y 312.491,Z 243.02,A -85,B 0,C 180,E1 -15790.709,E2 -15790.709} C_VEL
LIN {X 0,Y 312.509,Z 243.033,A -85,B 0,C 180,E1 -15794.199,E2 -15794.199} C_VEL
LIN {X 0,Y 312.551,Z 243.045,A -85,B 0,C 180,E1 -15797.905,E2 -15797.905} C_VEL
LIN {X 0,Y 312.555,Z 243.054,A -85,B 0,C 180,E1 -15801.905,E2 -15801.905} C_VEL
LIN {X 0,Y 312.503,Z 243.039,A -85,B 0,C 180,E1 -15805.791,E2 -15805.791} C_VEL
LIN {X 0,Y 312.521,Z 243.056,A -85,B 0,C 180,E1 -15808.855,E2 -15808.855} C_VEL
LIN {X 0,Y 312.571,Z 243.026,A -85,B 0,C 180,E1 -15811.825,E2 -15811.825} C_VEL
LIN {X 0,Y 312.582,Z 243.041,A -85,B 0,C 180,E1 -15814.711,E2 -15814.711} C_VEL
LIN {X 0,Y 312.535,Z 243.041,A -85,B 0,C 180,E1 -15818.913,E2 -15818.913} C_VEL
LIN {X 0,Y 312.636,Z 243.012,A -85,B 0,C 180,E1 -15821.657,E2 -15821.657} C_VEL
LIN {X 0,Y 312.692,Z 243.035,A -85,B 0,C 180,E1 -15825.687,E2 -15825.687} C_VEL
LIN {X 0,Y 312.697,Z 242.998,A -85,B 0,C 180,E1 -15829.642,E2 -15829.642} C_VEL
LIN {X 0,Y 312.852,Z 243.001,A -85,B 0,C 180,E1 -15832.255,E2 -15832.255} C_VEL
LIN {X 0,Y 312.714,Z 243.031,A -85,B 0,C 180,E1 -15834.843,E2 -15834.843} C_VEL
LIN {X 0,Y 312.718,Z 243.024,A -85,B 0,C 180,E1 -15836.324,E2 -15836.324} C_VEL
LIN {X 0,Y 312.188,Z 243.083,A -85,B 0,C 180,E1 -15837.402,E2 -15837.402} C_VEL
LIN {X 0,Y 309.455,Z 243.404,A -85,B 0,C 180,E1 -15839.16,E2 -15839.16} C_VEL
LIN {X 0,Y 307.051,Z 243.704,A -85,B 0,C 180,E1 -15840.585,E2 -15840.585} C_VEL
LIN {X 0,Y 305.992,Z 243.848,A -85,B 0,C 180,E1 -15841.688,E2 -15841.688} C_VEL
LIN {X 0,Y 305.895,Z 243.861,A -85,B 0,C 180,E1 -15842.061,E2 -15842.061} C_VEL
LIN {X 0,Y 305.797,Z 243.885,A -85,B 0,C 180,E1 -15846.599,E2 -15846.599} C_VEL
LIN {X 0,Y 305.694,Z 243.869,A -85,B 0,C 180,E1 -15849.262,E2 -15849.262} C_VEL
LIN {X 0,Y 305.588,Z 243.917,A -85,B 0,C 180,E1 -15853.297,E2 -15853.297} C_VEL
LIN {X 0,Y 305.555,Z 243.915,A -85,B 0,C 180,E1 -15856.023,E2 -15856.023} C_VEL
LIN {X 0,Y 305.548,Z 243.894,A -85,B 0,C 180,E1 -15859.43,E2 -15859.43} C_VEL
LIN {X 0,Y 305.491,Z 243.93,A -85,B 0,C 180,E1 -15863.042,E2 -15863.042} C_VEL
LIN {X 0,Y 305.526,Z 243.902,A -85,B 0,C 180,E1 -15866.219,E2 -15866.219} C_VEL
LIN {X 0,Y 305.489,Z 243.924,A -85,B 0,C 180,E1 -15869.048,E2 -15869.048} C_VEL
LIN {X 0,Y 305.444,Z 243.935,A -85,B 0,C 180,E1 -15871.953,E2 -15871.953} C_VEL
LIN {X 0,Y 305.462,Z 243.92,A -85,B 0,C 180,E1 -15875.114,E2 -15875.114} C_VEL
LIN {X 0,Y 305.467,Z 243.928,A -85,B 0,C 180,E1 -15878.533,E2 -15878.533} C_VEL
LIN {X 0,Y 305.457,Z 243.937,A -85,B 0,C 180,E1 -15882.586,E2 -15882.586} C_VEL
LIN {X 0,Y 305.427,Z 243.943,A -85,B 0,C 180,E1 -15886.345,E2 -15886.345} C_VEL
LIN {X 0,Y 305.46,Z 243.907,A -85,B 0,C 180,E1 -15889.893,E2 -15889.893} C_VEL
LIN {X 0,Y 305.486,Z 243.917,A -85,B 0,C 180,E1 -15893.632,E2 -15893.632} C_VEL
LIN {X 0,Y 305.521,Z 244.099,A -85,B 0,C 180,E1 -15895.118,E2 -15895.118} C_VEL
LIN {X 0,Y 307.134,Z 251.624,A -85,B 0,C 180,E1 -15898.244,E2 -15898.244} C_VEL
LIN {X 0,Y 308.645,Z 259.568,A -85,B 0,C 180,E1 -15901.433,E2 -15901.433} C_VEL
LIN {X 0,Y 309.173,Z 263.441,A -85,B 0,C 180,E1 -15902.959,E2 -15902.959} C_VEL
LIN {X 0,Y 309.08,Z 265.611,A -85,B 0,C 180,E1 -15903.669,E2 -15903.669} C_VEL
LIN {X 0,Y 311.433,Z 276.212,A -85,B 0,C 180,E1 -15904.198,E2 -15904.198} C_VEL
LIN {X 0,Y 316.387,Z 301.305,A -85,B 0,C 180,E1 -15905.242,E2 -15905.242} C_VEL
LIN {X 0,Y 317.597,Z 309.655,A -85,B 0,C 180,E1 -15905.545,E2 -15905.545} C_VEL
LIN {X 0,Y 316.091,Z 371.692,A -85,B 0,C 180,E1 -15906.972,E2 -15906.972} C_VEL
LIN {X 0,Y 315.456,Z 382.004,A -85,B 0,C 180,E1 -15907.356,E2 -15907.356} C_VEL
LIN {X 0,Y 314.689,Z 391.518,A -85,B 0,C 180,E1 -15907.86,E2 -15907.86} C_VEL
LIN {X 0,Y 313.637,Z 401.597,A -85,B 0,C 180,E1 -15908.56,E2 -15908.56} C_VEL
LIN {X 0,Y 312.494,Z 411.355,A -85,B 0,C 180,E1 -15909.427,E2 -15909.427} C_VEL
LIN {X 0,Y 311.115,Z 421.42,A -85,B 0,C 180,E1 -15910.537,E2 -15910.537} C_VEL
LIN {X 0,Y 309.373,Z 432.918,A -85,B 0,C 180,E1 -15912.141,E2 -15912.141} C_VEL
LIN {X 0,Y 308.141,Z 441.514,A -85,B 0,C 180,E1 -15913.662,E2 -15913.662} C_VEL
LIN {X 0,Y 307.024,Z 448.26,A -85,B 0,C 180,E1 -15915.077,E2 -15915.077} C_VEL
LIN {X 0,Y 305.935,Z 454.797,A -85,B 0,C 180,E1 -15916.719,E2 -15916.719} C_VEL
LIN {X 0,Y 305.204,Z 459.298,A -85,B 0,C 180,E1 -15918.039,E2 -15918.039} C_VEL
LIN {X 0,Y 304.456,Z 464.791,A -85,B 0,C 180,E1 -15920.03,E2 -15920.03} C_VEL
LIN {X 0,Y 303.958,Z 469.118,A -85,B 0,C 180,E1 -15922.026,E2 -15922.026} C_VEL
LIN {X 0,Y 303.743,Z 471.486,A -85,B 0,C 180,E1 -15923.357,E2 -15923.357} C_VEL
LIN {X 0,Y 303.64,Z 473.287,A -85,B 0,C 180,E1 -15924.688,E2 -15924.688} C_VEL
LIN {X 0,Y 303.603,Z 475.737,A -85,B 0,C 180,E1 -15927.346,E2 -15927.346} C_VEL
LIN {X 0,Y 303.566,Z 476.326,A -85,B 0,C 180,E1 -15928.673,E2 -15928.673} C_VEL
LIN {X 0,Y 303.566,Z 476.326,A -85,B 0,C 180,E1 -15931.327,E2 -15931.327} C_VEL
LIN {X 0,Y 303.603,Z 475.737,A -85,B 0,C 180,E1 -15932.654,E2 -15932.654} C_VEL
LIN {X 0,Y 303.62,Z 473.287,A -85,B 0,C 180,E1 -15935.313,E2 -15935.313} C_VEL
LIN {X 0,Y 303.841,Z 470.335,A -85,B 0,C 180,E1 -15937.309,E2 -15937.309} C_VEL
LIN {X 0,Y 304.267,Z 466.346,A -85,B 0,C 180,E1 -15939.305,E2 -15939.305} C_VEL
LIN {X 0,Y 304.962,Z 461.215,A -85,B 0,C 180,E1 -15941.296,E2 -15941.296} C_VEL
LIN {X 0,Y 305.729,Z 455.952,A -85,B 0,C 180,E1 -15942.952,E2 -15942.952} C_VEL
LIN {X 0,Y 306.774,Z 449.636,A -85,B 0,C 180,E1 -15944.596,E2 -15944.596} C_VEL
LIN {X 0,Y 307.747,Z 443.685,A -85,B 0,C 180,E1 -15945.905,E2 -15945.905} C_VEL
LIN {X 0,Y 308.757,Z 436.756,A -85,B 0,C 180,E1 -15947.212,E2 -15947.212} C_VEL
LIN {X 0,Y 310.02,Z 428.578,A -85,B 0,C 180,E1 -15948.504,E2 -15948.504} C_VEL
LIN {X 0,Y 311.311,Z 420.069,A -85,B 0,C 180,E1 -15949.622,E2 -15949.622} C_VEL
LIN {X 0,Y 312.488,Z 411.355,A -85,B 0,C 180,E1 -15950.574,E2 -15950.574} C_VEL
LIN {X 0,Y 313.646,Z 401.597,A -85,B 0,C 180,E1 -15951.44,E2 -15951.44} C_VEL
LIN {X 0,Y 314.726,Z 391.519,A -85,B 0,C 180,E1 -15952.137,E2 -15952.137} C_VEL
LIN {X 0,Y 315.504,Z 382.005,A -85,B 0,C 180,E1 -15952.64,E2 -15952.64} C_VEL
LIN {X 0,Y 316.071,Z 371.692,A -85,B 0,C 180,E1 -15953.029,E2 -15953.029} C_VEL
LIN {X 0,Y 317.55,Z 310.13,A -85,B 0,C 180,E1 -15954.447,E2 -15954.447} C_VEL
LIN {X 0,Y 316.717,Z 303.416,A -85,B 0,C 180,E1 -15954.679,E2 -15954.679} C_VEL
LIN {X 0,Y 312.508,Z 281.167,A -85,B 0,C 180,E1 -15955.584,E2 -15955.584} C_VEL
LIN {X 0,Y 309.106,Z 265.822,A -85,B 0,C 180,E1 -15956.304,E2 -15956.304} C_VEL
LIN {X 0,Y 309.148,Z 264.39,A -85,B 0,C 180,E1 -15956.679,E2 -15956.679} C_VEL
LIN {X 0,Y 308.938,Z 261.11,A -85,B 0,C 180,E1 -15957.951,E2 -15957.951} C_VEL
LIN {X 0,Y 306.974,Z 250.763,A -85,B 0,C 180,E1 -15962.102,E2 -15962.102} C_VEL
LIN {X 0,Y 305.518,Z 243.973,A -85,B 0,C 180,E1 -15964.97,E2 -15964.97} C_VEL
LIN {X 0,Y 305.469,Z 243.926,A -85,B 0,C 180,E1 -15968.532,E2 -15968.532} C_VEL
LIN {X 0,Y 305.457,Z 243.93,A -85,B 0,C 180,E1 -15972.585,E2 -15972.585} C_VEL
LIN {X 0,Y 305.427,Z 243.935,A -85,B 0,C 180,E1 -15976.344,E2 -15976.344} C_VEL
LIN {X 0,Y 305.46,Z 243.921,A -85,B 0,C 180,E1 -15979.892,E2 -15979.892} C_VEL
LIN {X 0,Y 305.482,Z 243.929,A -85,B 0,C 180,E1 -15983.631,E2 -15983.631} C_VEL
LIN {X 0,Y 305.466,Z 243.915,A -85,B 0,C 180,E1 -15986.483,E2 -15986.483} C_VEL
LIN {X 0,Y 305.459,Z 243.936,A -85,B 0,C 180,E1 -15989.59,E2 -15989.59} C_VEL
LIN {X 0,Y 305.497,Z 243.905,A -85,B 0,C 180,E1 -15992.606,E2 -15992.606} C_VEL
LIN {X 0,Y 305.508,Z 243.921,A -85,B 0,C 180,E1 -15995.538,E2 -15995.538} C_VEL
LIN {X 0,Y 305.507,Z 243.909,A -85,B 0,C 180,E1 -15999.813,E2 -15999.813} C_VEL
LIN {X 0,Y 305.546,Z 243.899,A -85,B 0,C 180,E1 -16002.601,E2 -16002.601} C_VEL
LIN {X 0,Y 305.627,Z 243.914,A -85,B 0,C 180,E1 -16005.347,E2 -16005.347} C_VEL
LIN {X 0,Y 305.624,Z 243.883,A -85,B 0,C 180,E1 -16009.399,E2 -16009.399} C_VEL
LIN {X 0,Y 305.764,Z 243.875,A -85,B 0,C 180,E1 -16012.072,E2 -16012.072} C_VEL
LIN {X 0,Y 305.675,Z 243.908,A -85,B 0,C 180,E1 -16014.723,E2 -16014.723} C_VEL
LIN {X 0,Y 305.955,Z 243.847,A -85,B 0,C 180,E1 -16018.683,E2 -16018.683} C_VEL
LIN {X 0,Y 305.955,Z 243.842,A -85,B 0,C 180,E1 -16021.316,E2 -16021.316} C_VEL
LIN {X 0,Y 305.685,Z 243.906,A -85,B 0,C 180,E1 -16025.276,E2 -16025.276} C_VEL
LIN {X 0,Y 305.795,Z 243.875,A -85,B 0,C 180,E1 -16027.925,E2 -16027.925} C_VEL
LIN {X 0,Y 305.602,Z 243.901,A -85,B 0,C 180,E1 -16031.944,E2 -16031.944} C_VEL
LIN {X 0,Y 305.636,Z 243.912,A -85,B 0,C 180,E1 -16035.034,E2 -16035.034} C_VEL
LIN {X 0,Y 305.578,Z 243.888,A -85,B 0,C 180,E1 -16038.782,E2 -16038.782} C_VEL
LIN {X 0,Y 305.484,Z 243.932,A -85,B 0,C 180,E1 -16043.039,E2 -16043.039} C_VEL
LIN {X 0,Y 305.523,Z 243.905,A -85,B 0,C 180,E1 -16046.218,E2 -16046.218} C_VEL
LIN {X 0,Y 305.493,Z 243.92,A -85,B 0,C 180,E1 -16049.049,E2 -16049.049} C_VEL
LIN {X 0,Y 305.442,Z 243.938,A -85,B 0,C 180,E1 -16051.951,E2 -16051.951} C_VEL
LIN {X 0,Y 305.459,Z 243.917,A -85,B 0,C 180,E1 -16055.113,E2 -16055.113} C_VEL
LIN {X 0,Y 305.489,Z 243.93,A -85,B 0,C 180,E1 -16058.538,E2 -16058.538} C_VEL
LIN {X 0,Y 305.512,Z 243.929,A -85,B 0,C 180,E1 -16062.598,E2 -16062.598} C_VEL
LIN {X 0,Y 305.465,Z 243.898,A -85,B 0,C 180,E1 -16066.352,E2 -16066.352} C_VEL
LIN {X 0,Y 305.459,Z 243.906,A -85,B 0,C 180,E1 -16069.893,E2 -16069.893} C_VEL
LIN {X 0,Y 305.493,Z 243.921,A -85,B 0,C 180,E1 -16073.263,E2 -16073.263} C_VEL
LIN {X 0,Y 305.461,Z 243.909,A -85,B 0,C 180,E1 -16076.483,E2 -16076.483} C_VEL
LIN {X 0,Y 305.454,Z 243.919,A -85,B 0,C 180,E1 -16079.59,E2 -16079.59} C_VEL
LIN {X 0,Y 305.528,Z 244.084,A -85,B 0,C 180,E1 -16082.989,E2 -16082.989} C_VEL
LIN {X 0,Y 305.764,Z 245.103,A -85,B 0,C 180,E1 -16083.25,E2 -16083.25} C_VEL
LIN {X 0,Y 309.589,Z 251.688,A -85,B 0,C 180,E1 -16083.846,E2 -16083.846} C_VEL
LIN {X 0,Y 314.965,Z 259.578,A -85,B 0,C 180,E1 -16084.681,E2 -16084.681} C_VEL
LIN {X 0,Y 321.523,Z 267.388,A -85,B 0,C 180,E1 -16085.752,E2 -16085.752} C_VEL
LIN {X 0,Y 326.495,Z 273.071,A -85,B 0,C 180,E1 -16086.657,E2 -16086.657} C_VEL
LIN {X 0,Y 331.237,Z 278.428,A -85,B 0,C 180,E1 -16087.584,E2 -16087.584} C_VEL
LIN {X 0,Y 337.794,Z 285.178,A -85,B 0,C 180,E1 -16088.948,E2 -16088.948} C_VEL
LIN {X 0,Y 344.299,Z 291.634,A -85,B 0,C 180,E1 -16090.401,E2 -16090.401} C_VEL
LIN {X 0,Y 347.95,Z 294.982,A -85,B 0,C 180,E1 -16091.26,E2 -16091.26} C_VEL
LIN {X 0,Y 353.194,Z 299.546,A -85,B 0,C 180,E1 -16092.579,E2 -16092.579} C_VEL
LIN {X 0,Y 359.548,Z 305.306,A -85,B 0,C 180,E1 -16094.358,E2 -16094.358} C_VEL
LIN {X 0,Y 364.237,Z 308.926,A -85,B 0,C 180,E1 -16095.799,E2 -16095.799} C_VEL
LIN {X 0,Y 368.573,Z 312.76,A -85,B 0,C 180,E1 -16097.311,E2 -16097.311} C_VEL
LIN {X 0,Y 372.511,Z 315.385,A -85,B 0,C 180,E1 -16098.827,E2 -16098.827} C_VEL
LIN {X 0,Y 374.583,Z 316.71,A -85,B 0,C 180,E1 -16099.7,E2 -16099.7} C_VEL
LIN {X 0,Y 377.882,Z 319.884,A -85,B 0,C 180,E1 -16101.376,E2 -16101.376} C_VEL
LIN {X 0,Y 380.706,Z 321.94,A -85,B 0,C 180,E1 -16103.09,E2 -16103.09} C_VEL
LIN {X 0,Y 383.172,Z 323.285,A -85,B 0,C 180,E1 -16105.011,E2 -16105.011} C_VEL
LIN {X 0,Y 384.859,Z 323.829,A -85,B 0,C 180,E1 -16106.86,E2 -16106.86} C_VEL
LIN {X 0,Y 385.794,Z 324.43,A -85,B 0,C 180,E1 -16108.956,E2 -16108.956} C_VEL
LIN {X 0,Y 385.946,Z 324.367,A -85,B 0,C 180,E1 -16110,E2 -16110} C_VEL
LIN {X 0,Y 385.654,Z 324.303,A -85,B 0,C 180,E1 -16111.566,E2 -16111.566} C_VEL
LIN {X 0,Y 384.854,Z 323.862,A -85,B 0,C 180,E1 -16113.14,E2 -16113.14} C_VEL
LIN {X 0,Y 383.172,Z 323.287,A -85,B 0,C 180,E1 -16114.989,E2 -16114.989} C_VEL
LIN {X 0,Y 380.706,Z 321.938,A -85,B 0,C 180,E1 -16116.91,E2 -16116.91} C_VEL
LIN {X 0,Y 377.565,Z 319.646,A -85,B 0,C 180,E1 -16118.792,E2 -16118.792} C_VEL
LIN {X 0,Y 373.598,Z 315.957,A -85,B 0,C 180,E1 -16120.732,E2 -16120.732} C_VEL
LIN {X 0,Y 369.701,Z 313.563,A -85,B 0,C 180,E1 -16122.277,E2 -16122.277} C_VEL
LIN {X 0,Y 365.467,Z 310.1,A -85,B 0,C 180,E1 -16123.787,E2 -16123.787} C_VEL
LIN {X 0,Y 362.243,Z 307.264,A -85,B 0,C 180,E1 -16124.835,E2 -16124.835} C_VEL
LIN {X 0,Y 357.096,Z 303.18,A -85,B 0,C 180,E1 -16126.35,E2 -16126.35} C_VEL
LIN {X 0,Y 353.196,Z 299.52,A -85,B 0,C 180,E1 -16127.421,E2 -16127.421} C_VEL
LIN {X 0,Y 348.233,Z 295.28,A -85,B 0,C 180,E1 -16128.671,E2 -16128.671} C_VEL
LIN {X 0,Y 344.3,Z 291.618,A -85,B 0,C 180,E1 -16129.599,E2 -16129.599} C_VEL
LIN {X 0,Y 339.417,Z 286.716,A -85,B 0,C 180,E1 -16130.71,E2 -16130.71} C_VEL
LIN {X 0,Y 333.452,Z 280.679,A -85,B 0,C 180,E1 -16131.974,E2 -16131.974} C_VEL
LIN {X 0,Y 327.607,Z 274.426,A -85,B 0,C 180,E1 -16133.128,E2 -16133.128} C_VEL
LIN {X 0,Y 321.997,Z 267.927,A -85,B 0,C 180,E1 -16134.165,E2 -16134.165} C_VEL
LIN {X 0,Y 317.662,Z 262.765,A -85,B 0,C 180,E1 -16134.896,E2 -16134.896} C_VEL
LIN {X 0,Y 313.561,Z 257.596,A -85,B 0,C 180,E1 -16135.539,E2 -16135.539} C_VEL
LIN {X 0,Y 308.173,Z 249.646,A -85,B 0,C 180,E1 -16136.352,E2 -16136.352} C_VEL
LIN {X 0,Y 305.762,Z 245.11,A -85,B 0,C 180,E1 -16136.749,E2 -16136.749} C_VEL
LIN {X 0,Y 305.528,Z 244.086,A -85,B 0,C 180,E1 -16137.01,E2 -16137.01} C_VEL
LIN {X 0,Y 305.454,Z 243.919,A -85,B 0,C 180,E1 -16140.41,E2 -16140.41} C_VEL
LIN {X 0,Y 305.461,Z 243.904,A -85,B 0,C 180,E1 -16144.079,E2 -16144.079} C_VEL
LIN {X 0,Y 305.493,Z 243.921,A -85,B 0,C 180,E1 -16146.737,E2 -16146.737} C_VEL
LIN {X 0,Y 305.459,Z 243.906,A -85,B 0,C 180,E1 -16150.107,E2 -16150.107} C_VEL
LIN {X 0,Y 305.465,Z 243.898,A -85,B 0,C 180,E1 -16153.648,E2 -16153.648} C_VEL
LIN {X 0,Y 305.512,Z 243.929,A -85,B 0,C 180,E1 -16157.402,E2 -16157.402} C_VEL
LIN {X 0,Y 305.517,Z 243.928,A -85,B 0,C 180,E1 -16161.605,E2 -16161.605} C_VEL
LIN {X 0,Y 305.459,Z 243.917,A -85,B 0,C 180,E1 -16164.887,E2 -16164.887} C_VEL
LIN {X 0,Y 305.449,Z 243.938,A -85,B 0,C 180,E1 -16168.355,E2 -16168.355} C_VEL
LIN {X 0,Y 305.518,Z 243.913,A -85,B 0,C 180,E1 -16171.114,E2 -16171.114} C_VEL
LIN {X 0,Y 305.563,Z 243.905,A -85,B 0,C 180,E1 -16174.088,E2 -16174.088} C_VEL
LIN {X 0,Y 305.479,Z 243.925,A -85,B 0,C 180,E1 -16178.402,E2 -16178.402} C_VEL
LIN {X 0,Y 305.578,Z 243.888,A -85,B 0,C 180,E1 -16181.218,E2 -16181.218} C_VEL
LIN {X 0,Y 305.648,Z 243.914,A -85,B 0,C 180,E1 -16185.35,E2 -16185.35} C_VEL
LIN {X 0,Y 305.634,Z 243.879,A -85,B 0,C 180,E1 -16189.4,E2 -16189.4} C_VEL
LIN {X 0,Y 305.795,Z 243.875,A -85,B 0,C 180,E1 -16192.075,E2 -16192.075} C_VEL
LIN {X 0,Y 305.685,Z 243.906,A -85,B 0,C 180,E1 -16194.724,E2 -16194.724} C_VEL
LIN {X 0,Y 305.955,Z 243.842,A -85,B 0,C 180,E1 -16198.684,E2 -16198.684} C_VEL
LIN {X 0,Y 305.955,Z 243.847,A -85,B 0,C 180,E1 -16201.317,E2 -16201.317} C_VEL
LIN {X 0,Y 305.895,Z 243.861,A -85,B 0,C 180,E1 -16202.061,E2 -16202.061} C_VEL
LIN {X 0,Y 305.184,Z 243.965,A -85,B 0,C 180,E1 -16203.158,E2 -16203.158} C_VEL
LIN {X 0,Y 302.265,Z 244.336,A -85,B 0,C 180,E1 -16204.943,E2 -16204.943} C_VEL
LIN {X 0,Y 299.817,Z 244.633,A -85,B 0,C 180,E1 -16206.39,E2 -16206.39} C_VEL
LIN {X 0,Y 298.783,Z 244.748,A -85,B 0,C 180,E1 -16207.513,E2 -16207.513} C_VEL
LIN {X 0,Y 298.706,Z 244.751,A -85,B 0,C 180,E1 -16207.893,E2 -16207.893} C_VEL
LIN {X 0,Y 298.55,Z 244.784,A -85,B 0,C 180,E1 -16212.232,E2 -16212.232} C_VEL
LIN {X 0,Y 298.55,Z 244.79,A -85,B 0,C 180,E1 -16215.17,E2 -16215.17} C_VEL
LIN {X 0,Y 298.509,Z 244.769,A -85,B 0,C 180,E1 -16219.246,E2 -16219.246} C_VEL
LIN {X 0,Y 298.458,Z 244.804,A -85,B 0,C 180,E1 -16223.598,E2 -16223.598} C_VEL
LIN {X 0,Y 298.485,Z 244.777,A -85,B 0,C 180,E1 -16226.576,E2 -16226.576} C_VEL
LIN {X 0,Y 298.418,Z 244.809,A -85,B 0,C 180,E1 -16229.642,E2 -16229.642} C_VEL
LIN {X 0,Y 298.396,Z 244.801,A -85,B 0,C 180,E1 -16232.801,E2 -16232.801} C_VEL
LIN {X 0,Y 298.447,Z 244.811,A -85,B 0,C 180,E1 -16236.808,E2 -16236.808} C_VEL
LIN {X 0,Y 298.41,Z 244.801,A -85,B 0,C 180,E1 -16239.487,E2 -16239.487} C_VEL
LIN {X 0,Y 298.4,Z 244.813,A -85,B 0,C 180,E1 -16243.104,E2 -16243.104} C_VEL
LIN {X 0,Y 298.405,Z 244.814,A -85,B 0,C 180,E1 -16246.921,E2 -16246.921} C_VEL
LIN {X 0,Y 298.417,Z 244.794,A -85,B 0,C 180,E1 -16251.004,E2 -16251.004} C_VEL
LIN {X 0,Y 298.47,Z 244.892,A -85,B 0,C 180,E1 -16254.549,E2 -16254.549} C_VEL
LIN {X 0,Y 299.599,Z 250.38,A -85,B 0,C 180,E1 -16256.948,E2 -16256.948} C_VEL
LIN {X 0,Y 301.429,Z 259.358,A -85,B 0,C 180,E1 -16260.684,E2 -16260.684} C_VEL
LIN {X 0,Y 302.233,Z 265.018,A -85,B 0,C 180,E1 -16262.941,E2 -16262.941} C_VEL
LIN {X 0,Y 302.472,Z 266.415,A -85,B 0,C 180,E1 -16263.113,E2 -16263.113} C_VEL
LIN {X 0,Y 307.573,Z 289.527,A -85,B 0,C 180,E1 -16264.191,E2 -16264.191} C_VEL
LIN {X 0,Y 310.999,Z 309.101,A -85,B 0,C 180,E1 -16264.982,E2 -16264.982} C_VEL
LIN {X 0,Y 309.996,Z 358.96,A -85,B 0,C 180,E1 -16266.138,E2 -16266.138} C_VEL
LIN {X 0,Y 309.33,Z 376.543,A -85,B 0,C 180,E1 -16266.616,E2 -16266.616} C_VEL
LIN {X 0,Y 308.345,Z 388.749,A -85,B 0,C 180,E1 -16267.203,E2 -16267.203} C_VEL
LIN {X 0,Y 307.278,Z 399.391,A -85,B 0,C 180,E1 -16267.917,E2 -16267.917} C_VEL
LIN {X 0,Y 306.033,Z 409.529,A -85,B 0,C 180,E1 -16268.796,E2 -16268.796} C_VEL
LIN {X 0,Y 304.837,Z 418.525,A -85,B 0,C 180,E1 -16269.768,E2 -16269.768} C_VEL
LIN {X 0,Y 303.433,Z 427.249,A -85,B 0,C 180,E1 -16270.904,E2 -16270.904} C_VEL
LIN {X 0,Y 302.281,Z 434.644,A -85,B 0,C 180,E1 -16272.058,E2 -16272.058} C_VEL
LIN {X 0,Y 301.211,Z 441.948,A -85,B 0,C 180,E1 -16273.41,E2 -16273.41} C_VEL
LIN {X 0,Y 300.119,Z 448.066,A -85,B 0,C 180,E1 -16274.725,E2 -16274.725} C_VEL
LIN {X 0,Y 299.001,Z 454.603,A -85,B 0,C 180,E1 -16276.406,E2 -16276.406} C_VEL
LIN {X 0,Y 298.227,Z 459.104,A -85,B 0,C 180,E1 -16277.755,E2 -16277.755} C_VEL
LIN {X 0,Y 297.437,Z 464.598,A -85,B 0,C 180,E1 -16279.793,E2 -16279.793} C_VEL
LIN {X 0,Y 296.899,Z 468.924,A -85,B 0,C 180,E1 -16281.835,E2 -16281.835} C_VEL
LIN {X 0,Y 296.69,Z 471.293,A -85,B 0,C 180,E1 -16283.198,E2 -16283.198} C_VEL
LIN {X 0,Y 296.554,Z 473.094,A -85,B 0,C 180,E1 -16284.56,E2 -16284.56} C_VEL
LIN {X 0,Y 296.528,Z 475.545,A -85,B 0,C 180,E1 -16287.283,E2 -16287.283} C_VEL
LIN {X 0,Y 296.486,Z 476.133,A -85,B 0,C 180,E1 -16288.642,E2 -16288.642} C_VEL
LIN {X 0,Y 296.486,Z 476.133,A -85,B 0,C 180,E1 -16291.358,E2 -16291.358} C_VEL
LIN {X 0,Y 296.528,Z 475.545,A -85,B 0,C 180,E1 -16292.717,E2 -16292.717} C_VEL
LIN {X 0,Y 296.549,Z 473.003,A -85,B 0,C 180,E1 -16295.509,E2 -16295.509} C_VEL
LIN {X 0,Y 296.79,Z 470.142,A -85,B 0,C 180,E1 -16297.483,E2 -16297.483} C_VEL
LIN {X 0,Y 297.239,Z 466.152,A -85,B 0,C 180,E1 -16299.527,E2 -16299.527} C_VEL
LIN {X 0,Y 297.953,Z 461.021,A -85,B 0,C 180,E1 -16301.566,E2 -16301.566} C_VEL
LIN {X 0,Y 298.793,Z 455.758,A -85,B 0,C 180,E1 -16303.258,E2 -16303.258} C_VEL
LIN {X 0,Y 299.866,Z 449.442,A -85,B 0,C 180,E1 -16304.94,E2 -16304.94} C_VEL
LIN {X 0,Y 300.918,Z 443.492,A -85,B 0,C 180,E1 -16306.276,E2 -16306.276} C_VEL
LIN {X 0,Y 301.966,Z 436.563,A -85,B 0,C 180,E1 -16307.612,E2 -16307.612} C_VEL
LIN {X 0,Y 303.284,Z 428.385,A -85,B 0,C 180,E1 -16308.93,E2 -16308.93} C_VEL
LIN {X 0,Y 304.619,Z 419.876,A -85,B 0,C 180,E1 -16310.071,E2 -16310.071} C_VEL
LIN {X 0,Y 305.822,Z 411.161,A -85,B 0,C 180,E1 -16311.043,E2 -16311.043} C_VEL
LIN {X 0,Y 307.047,Z 401.405,A -85,B 0,C 180,E1 -16311.924,E2 -16311.924} C_VEL
LIN {X 0,Y 308.049,Z 392.614,A -85,B 0,C 180,E1 -16312.555,E2 -16312.555} C_VEL
LIN {X 0,Y 308.886,Z 382.686,A -85,B 0,C 180,E1 -16313.109,E2 -16313.109} C_VEL
LIN {X 0,Y 309.514,Z 372.831,A -85,B 0,C 180,E1 -16313.502,E2 -16313.502} C_VEL
LIN {X 0,Y 310.215,Z 348.025,A -85,B 0,C 180,E1 -16314.116,E2 -16314.116} C_VEL
LIN {X 0,Y 311.004,Z 308.92,A -85,B 0,C 180,E1 -16315.022,E2 -16315.022} C_VEL
LIN {X 0,Y 306.837,Z 285.8,A -85,B 0,C 180,E1 -16315.97,E2 -16315.97} C_VEL
LIN {X 0,Y 302.322,Z 265.848,A -85,B 0,C 180,E1 -16316.922,E2 -16316.922} C_VEL
LIN {X 0,Y 302.228,Z 265.016,A -85,B 0,C 180,E1 -16317.059,E2 -16317.059} C_VEL
LIN {X 0,Y 301.761,Z 261.304,A -85,B 0,C 180,E1 -16318.518,E2 -16318.518} C_VEL
LIN {X 0,Y 300.283,Z 253.572,A -85,B 0,C 180,E1 -16321.707,E2 -16321.707} C_VEL
LIN {X 0,Y 298.471,Z 244.867,A -85,B 0,C 180,E1 -16325.452,E2 -16325.452} C_VEL
LIN {X 0,Y 298.411,Z 244.789,A -85,B 0,C 180,E1 -16329.486,E2 -16329.486} C_VEL
LIN {X 0,Y 298.401,Z 244.814,A -85,B 0,C 180,E1 -16333.103,E2 -16333.103} C_VEL
LIN {X 0,Y 298.405,Z 244.812,A -85,B 0,C 180,E1 -16336.92,E2 -16336.92} C_VEL
LIN {X 0,Y 298.416,Z 244.803,A -85,B 0,C 180,E1 -16341.003,E2 -16341.003} C_VEL
LIN {X 0,Y 298.419,Z 244.806,A -85,B 0,C 180,E1 -16343.929,E2 -16343.929} C_VEL
LIN {X 0,Y 298.395,Z 244.811,A -85,B 0,C 180,E1 -16347.983,E2 -16347.983} C_VEL
LIN {X 0,Y 298.45,Z 244.789,A -85,B 0,C 180,E1 -16351.902,E2 -16351.902} C_VEL
LIN {X 0,Y 298.483,Z 244.79,A -85,B 0,C 180,E1 -16354.923,E2 -16354.923} C_VEL
LIN {X 0,Y 298.443,Z 244.792,A -85,B 0,C 180,E1 -16359.314,E2 -16359.314} C_VEL
LIN {X 0,Y 298.508,Z 244.77,A -85,B 0,C 180,E1 -16362.177,E2 -16362.177} C_VEL
LIN {X 0,Y 298.586,Z 244.787,A -85,B 0,C 180,E1 -16364.994,E2 -16364.994} C_VEL
LIN {X 0,Y 298.583,Z 244.761,A -85,B 0,C 180,E1 -16369.146,E2 -16369.146} C_VEL
LIN {X 0,Y 298.712,Z 244.749,A -85,B 0,C 180,E1 -16371.884,E2 -16371.884} C_VEL
LIN {X 0,Y 298.643,Z 244.783,A -85,B 0,C 180,E1 -16374.598,E2 -16374.598} C_VEL
LIN {X 0,Y 298.921,Z 244.722,A -85,B 0,C 180,E1 -16378.652,E2 -16378.652} C_VEL
LIN {X 0,Y 298.922,Z 244.717,A -85,B 0,C 180,E1 -16381.346,E2 -16381.346} C_VEL
LIN {X 0,Y 298.786,Z 244.759,A -85,B 0,C 180,E1 -16386.753,E2 -16386.753} C_VEL
LIN {X 0,Y 298.634,Z 244.749,A -85,B 0,C 180,E1 -16389.481,E2 -16389.481} C_VEL
LIN {X 0,Y 298.551,Z 244.793,A -85,B 0,C 180,E1 -16393.615,E2 -16393.615} C_VEL
LIN {X 0,Y 298.547,Z 244.788,A -85,B 0,C 180,E1 -16396.408,E2 -16396.408} C_VEL
LIN {X 0,Y 298.496,Z 244.771,A -85,B 0,C 180,E1 -16399.646,E2 -16399.646} C_VEL
LIN {X 0,Y 298.426,Z 244.811,A -85,B 0,C 180,E1 -16403.599,E2 -16403.599} C_VEL
LIN {X 0,Y 298.481,Z 244.778,A -85,B 0,C 180,E1 -16406.574,E2 -16406.574} C_VEL
LIN {X 0,Y 298.418,Z 244.806,A -85,B 0,C 180,E1 -16409.64,E2 -16409.64} C_VEL
LIN {X 0,Y 298.393,Z 244.808,A -85,B 0,C 180,E1 -16412.8,E2 -16412.8} C_VEL
LIN {X 0,Y 298.467,Z 244.807,A -85,B 0,C 180,E1 -16416.813,E2 -16416.813} C_VEL
LIN {X 0,Y 298.45,Z 244.793,A -85,B 0,C 180,E1 -16421.249,E2 -16421.249} C_VEL
LIN {X 0,Y 298.413,Z 244.799,A -85,B 0,C 180,E1 -16425.046,E2 -16425.046} C_VEL
LIN {X 0,Y 298.388,Z 244.769,A -85,B 0,C 180,E1 -16428.911,E2 -16428.911} C_VEL
LIN {X 0,Y 298.441,Z 244.811,A -85,B 0,C 180,E1 -16432.246,E2 -16432.246} C_VEL
LIN {X 0,Y 298.404,Z 244.781,A -85,B 0,C 180,E1 -16435.581,E2 -16435.581} C_VEL
LIN {X 0,Y 298.388,Z 244.812,A -85,B 0,C 180,E1 -16438.791,E2 -16438.791} C_VEL
LIN {X 0,Y 298.479,Z 244.969,A -85,B 0,C 180,E1 -16442.324,E2 -16442.324} C_VEL
LIN {X 0,Y 298.787,Z 246.114,A -85,B 0,C 180,E1 -16442.597,E2 -16442.597} C_VEL
LIN {X 0,Y 303.453,Z 254.678,A -85,B 0,C 180,E1 -16443.297,E2 -16443.297} C_VEL
LIN {X 0,Y 310.527,Z 264.723,A -85,B 0,C 180,E1 -16444.295,E2 -16444.295} C_VEL
LIN {X 0,Y 317.259,Z 272.572,A -85,B 0,C 180,E1 -16445.324,E2 -16445.324} C_VEL
LIN {X 0,Y 322.931,Z 278.827,A -85,B 0,C 180,E1 -16446.276,E2 -16446.276} C_VEL
LIN {X 0,Y 328.017,Z 284.384,A -85,B 0,C 180,E1 -16447.222,E2 -16447.222} C_VEL
LIN {X 0,Y 335.007,Z 291.426,A -85,B 0,C 180,E1 -16448.625,E2 -16448.625} C_VEL
LIN {X 0,Y 341.637,Z 297.901,A -85,B 0,C 180,E1 -16450.065,E2 -16450.065} C_VEL
LIN {X 0,Y 348.766,Z 304.354,A -85,B 0,C 180,E1 -16451.751,E2 -16451.751} C_VEL
LIN {X 0,Y 353.428,Z 308.21,A -85,B 0,C 180,E1 -16452.936,E2 -16452.936} C_VEL
LIN {X 0,Y 358.648,Z 312.715,A -85,B 0,C 180,E1 -16454.399,E2 -16454.399} C_VEL
LIN {X 0,Y 362.73,Z 315.895,A -85,B 0,C 180,E1 -16455.638,E2 -16455.638} C_VEL
LIN {X 0,Y 367.469,Z 319.877,A -85,B 0,C 180,E1 -16457.261,E2 -16457.261} C_VEL
LIN {X 0,Y 371.532,Z 322.464,A -85,B 0,C 180,E1 -16458.809,E2 -16458.809} C_VEL
LIN {X 0,Y 373.558,Z 323.939,A -85,B 0,C 180,E1 -16459.672,E2 -16459.672} C_VEL
LIN {X 0,Y 377.053,Z 327.109,A -85,B 0,C 180,E1 -16461.424,E2 -16461.424} C_VEL
LIN {X 0,Y 380.082,Z 329.161,A -85,B 0,C 180,E1 -16463.274,E2 -16463.274} C_VEL
LIN {X 0,Y 382.282,Z 330.331,A -85,B 0,C 180,E1 -16464.999,E2 -16464.999} C_VEL
LIN {X 0,Y 383.984,Z 330.854,A -85,B 0,C 180,E1 -16466.852,E2 -16466.852} C_VEL
LIN {X 0,Y 384.932,Z 331.473,A -85,B 0,C 180,E1 -16468.954,E2 -16468.954} C_VEL
LIN {X 0,Y 385.081,Z 331.414,A -85,B 0,C 180,E1 -16470,E2 -16470} C_VEL
LIN {X 0,Y 384.785,Z 331.351,A -85,B 0,C 180,E1 -16471.57,E2 -16471.57} C_VEL
LIN {X 0,Y 383.98,Z 330.887,A -85,B 0,C 180,E1 -16473.148,E2 -16473.148} C_VEL
LIN {X 0,Y 382.282,Z 330.334,A -85,B 0,C 180,E1 -16475.001,E2 -16475.001} C_VEL
LIN {X 0,Y 379.791,Z 328.992,A -85,B 0,C 180,E1 -16476.927,E2 -16476.927} C_VEL
LIN {X 0,Y 376.551,Z 326.736,A -85,B 0,C 180,E1 -16478.839,E2 -16478.839} C_VEL
LIN {X 0,Y 372.814,Z 323.209,A -85,B 0,C 180,E1 -16480.664,E2 -16480.664} C_VEL
LIN {X 0,Y 368.428,Z 320.566,A -85,B 0,C 180,E1 -16482.386,E2 -16482.386} C_VEL
LIN {X 0,Y 364.116,Z 317.136,A -85,B 0,C 180,E1 -16483.899,E2 -16483.899} C_VEL
LIN {X 0,Y 359.982,Z 313.677,A -85,B 0,C 180,E1 -16485.208,E2 -16485.208} C_VEL
LIN {X 0,Y 354.506,Z 309.282,A -85,B 0,C 180,E1 -16486.764,E2 -16486.764} C_VEL
LIN {X 0,Y 350.409,Z 305.628,A -85,B 0,C 180,E1 -16487.849,E2 -16487.849} C_VEL
LIN {X 0,Y 345.169,Z 301.104,A -85,B 0,C 180,E1 -16489.127,E2 -16489.127} C_VEL
LIN {X 0,Y 337.919,Z 294.404,A -85,B 0,C 180,E1 -16490.749,E2 -16490.749} C_VEL
LIN {X 0,Y 330.266,Z 286.71,A -85,B 0,C 180,E1 -16492.336,E2 -16492.336} C_VEL
LIN {X 0,Y 323.726,Z 279.782,A -85,B 0,C 180,E1 -16493.574,E2 -16493.574} C_VEL
LIN {X 0,Y 316.13,Z 271.425,A -85,B 0,C 180,E1 -16494.852,E2 -16494.852} C_VEL
LIN {X 0,Y 309.11,Z 262.811,A -85,B 0,C 180,E1 -16495.909,E2 -16495.909} C_VEL
LIN {X 0,Y 302.671,Z 253.413,A -85,B 0,C 180,E1 -16496.811,E2 -16496.811} C_VEL
LIN {X 0,Y 298.712,Z 245.914,A -85,B 0,C 180,E1 -16497.429,E2 -16497.429} C_VEL
LIN {X 0,Y 298.487,Z 244.901,A -85,B 0,C 180,E1 -16497.727,E2 -16497.727} C_VEL
LIN {X 0,Y 298.391,Z 244.817,A -85,B 0,C 180,E1 -16502.017,E2 -16502.017} C_VEL
LIN {X 0,Y 298.428,Z 244.789,A -85,B 0,C 180,E1 -16506.068,E2 -16506.068} C_VEL
LIN {X 0,Y 298.415,Z 244.796,A -85,B 0,C 180,E1 -16509.485,E2 -16509.485} C_VEL
LIN {X 0,Y 298.422,Z 244.766,A -85,B 0,C 180,E1 -16513.109,E2 -16513.109} C_VEL
LIN {X 0,Y 298.464,Z 244.806,A -85,B 0,C 180,E1 -16516.933,E2 -16516.933} C_VEL
LIN {X 0,Y 298.433,Z 244.808,A -85,B 0,C 180,E1 -16520.999,E2 -16520.999} C_VEL
LIN {X 0,Y 298.431,Z 244.801,A -85,B 0,C 180,E1 -16523.933,E2 -16523.933} C_VEL
LIN {X 0,Y 298.393,Z 244.815,A -85,B 0,C 180,E1 -16527.984,E2 -16527.984} C_VEL
LIN {X 0,Y 298.45,Z 244.783,A -85,B 0,C 180,E1 -16531.904,E2 -16531.904} C_VEL
LIN {X 0,Y 298.479,Z 244.798,A -85,B 0,C 180,E1 -16534.924,E2 -16534.924} C_VEL
LIN {X 0,Y 298.435,Z 244.789,A -85,B 0,C 180,E1 -16539.315,E2 -16539.315} C_VEL
LIN {X 0,Y 298.533,Z 244.774,A -85,B 0,C 180,E1 -16542.18,E2 -16542.18} C_VEL
LIN {X 0,Y 298.592,Z 244.79,A -85,B 0,C 180,E1 -16544.996,E2 -16544.996} C_VEL
LIN {X 0,Y 298.59,Z 244.758,A -85,B 0,C 180,E1 -16549.147,E2 -16549.147} C_VEL
LIN {X 0,Y 298.739,Z 244.75,A -85,B 0,C 180,E1 -16551.886,E2 -16551.886} C_VEL
LIN {X 0,Y 298.656,Z 244.782,A -85,B 0,C 180,E1 -16554.6,E2 -16554.6} C_VEL
LIN {X 0,Y 298.922,Z 244.717,A -85,B 0,C 180,E1 -16558.654,E2 -16558.654} C_VEL
LIN {X 0,Y 298.921,Z 244.722,A -85,B 0,C 180,E1 -16561.348,E2 -16561.348} C_VEL
LIN {X 0,Y 298.643,Z 244.783,A -85,B 0,C 180,E1 -16565.402,E2 -16565.402} C_VEL
LIN {X 0,Y 298.706,Z 244.751,A -85,B 0,C 180,E1 -16567.893,E2 -16567.893} C_VEL
LIN {X 0,Y 298.032,Z 244.83,A -85,B 0,C 180,E1 -16569.017,E2 -16569.017} C_VEL
LIN {X 0,Y 295.089,Z 245.199,A -85,B 0,C 180,E1 -16570.844,E2 -16570.844} C_VEL
LIN {X 0,Y 292.607,Z 245.524,A -85,B 0,C 180,E1 -16572.328,E2 -16572.328} C_VEL
LIN {X 0,Y 291.576,Z 245.662,A -85,B 0,C 180,E1 -16573.479,E2 -16573.479} C_VEL
LIN {X 0,Y 291.511,Z 245.668,A -85,B 0,C 180,E1 -16573.869,E2 -16573.869} C_VEL
LIN {X 0,Y 291.443,Z 245.659,A -85,B 0,C 180,E1 -16576.821,E2 -16576.821} C_VEL
LIN {X 0,Y 291.451,Z 245.653,A -85,B 0,C 180,E1 -16579.876,E2 -16579.876} C_VEL
LIN {X 0,Y 291.4,Z 245.682,A -85,B 0,C 180,E1 -16584.206,E2 -16584.206} C_VEL
LIN {X 0,Y 291.416,Z 245.657,A -85,B 0,C 180,E1 -16587.273,E2 -16587.273} C_VEL
LIN {X 0,Y 291.335,Z 245.696,A -85,B 0,C 180,E1 -16590.438,E2 -16590.438} C_VEL
LIN {X 0,Y 291.345,Z 245.672,A -85,B 0,C 180,E1 -16593.699,E2 -16593.699} C_VEL
LIN {X 0,Y 291.382,Z 245.689,A -85,B 0,C 180,E1 -16597.256,E2 -16597.256} C_VEL
LIN {X 0,Y 291.336,Z 245.682,A -85,B 0,C 180,E1 -16600.643,E2 -16600.643} C_VEL
LIN {X 0,Y 291.292,Z 245.691,A -85,B 0,C 180,E1 -16604.403,E2 -16604.403} C_VEL
LIN {X 0,Y 291.328,Z 245.673,A -85,B 0,C 180,E1 -16608.405,E2 -16608.405} C_VEL
LIN {X 0,Y 291.366,Z 245.674,A -85,B 0,C 180,E1 -16611.161,E2 -16611.161} C_VEL
LIN {X 0,Y 291.407,Z 245.751,A -85,B 0,C 180,E1 -16613.995,E2 -16613.995} C_VEL
LIN {X 0,Y 292.184,Z 249.469,A -85,B 0,C 180,E1 -16615.714,E2 -16615.714} C_VEL
LIN {X 0,Y 293.921,Z 258.017,A -85,B 0,C 180,E1 -16619.408,E2 -16619.408} C_VEL
LIN {X 0,Y 295.227,Z 265.046,A -85,B 0,C 180,E1 -16622.299,E2 -16622.299} C_VEL
LIN {X 0,Y 296.274,Z 268.488,A -85,B 0,C 180,E1 -16622.578,E2 -16622.578} C_VEL
LIN {X 0,Y 300.854,Z 289.053,A -85,B 0,C 180,E1 -16623.564,E2 -16623.564} C_VEL
LIN {X 0,Y 304.597,Z 310.131,A -85,B 0,C 180,E1 -16624.45,E2 -16624.45} C_VEL
LIN {X 0,Y 303.098,Z 371.308,A -85,B 0,C 180,E1 -16625.924,E2 -16625.924} C_VEL
LIN {X 0,Y 302.422,Z 381.619,A -85,B 0,C 180,E1 -16626.322,E2 -16626.322} C_VEL
LIN {X 0,Y 301.597,Z 391.133,A -85,B 0,C 180,E1 -16626.844,E2 -16626.844} C_VEL
LIN {X 0,Y 300.471,Z 401.212,A -85,B 0,C 180,E1 -16627.571,E2 -16627.571} C_VEL
LIN {X 0,Y 299.198,Z 410.968,A -85,B 0,C 180,E1 -16628.468,E2 -16628.468} C_VEL
LIN {X 0,Y 297.765,Z 421.034,A -85,B 0,C 180,E1 -16629.627,E2 -16629.627} C_VEL
LIN {X 0,Y 295.811,Z 432.53,A -85,B 0,C 180,E1 -16631.292,E2 -16631.292} C_VEL
LIN {X 0,Y 294.543,Z 440.853,A -85,B 0,C 180,E1 -16632.825,E2 -16632.825} C_VEL
LIN {X 0,Y 293.226,Z 447.872,A -85,B 0,C 180,E1 -16634.357,E2 -16634.357} C_VEL
LIN {X 0,Y 292.071,Z 454.409,A -85,B 0,C 180,E1 -16636.077,E2 -16636.077} C_VEL
LIN {X 0,Y 291.259,Z 458.91,A -85,B 0,C 180,E1 -16637.457,E2 -16637.457} C_VEL
LIN {X 0,Y 290.433,Z 464.404,A -85,B 0,C 180,E1 -16639.544,E2 -16639.544} C_VEL
LIN {X 0,Y 289.857,Z 468.731,A -85,B 0,C 180,E1 -16641.635,E2 -16641.635} C_VEL
LIN {X 0,Y 289.609,Z 471.1,A -85,B 0,C 180,E1 -16643.031,E2 -16643.031} C_VEL
LIN {X 0,Y 289.457,Z 473.066,A -85,B 0,C 180,E1 -16644.555,E2 -16644.555} C_VEL
LIN {X 0,Y 289.432,Z 475.352,A -85,B 0,C 180,E1 -16647.216,E2 -16647.216} C_VEL
LIN {X 0,Y 289.408,Z 475.941,A -85,B 0,C 180,E1 -16648.608,E2 -16648.608} C_VEL
LIN {X 0,Y 289.408,Z 475.941,A -85,B 0,C 180,E1 -16651.392,E2 -16651.392} C_VEL
LIN {X 0,Y 289.431,Z 475.352,A -85,B 0,C 180,E1 -16652.784,E2 -16652.784} C_VEL
LIN {X 0,Y 289.479,Z 472.901,A -85,B 0,C 180,E1 -16655.573,E2 -16655.573} C_VEL
LIN {X 0,Y 289.721,Z 469.949,A -85,B 0,C 180,E1 -16657.667,E2 -16657.667} C_VEL
LIN {X 0,Y 290.196,Z 465.958,A -85,B 0,C 180,E1 -16659.76,E2 -16659.76} C_VEL
LIN {X 0,Y 290.963,Z 460.827,A -85,B 0,C 180,E1 -16661.848,E2 -16661.848} C_VEL
LIN {X 0,Y 291.868,Z 455.565,A -85,B 0,C 180,E1 -16663.578,E2 -16663.578} C_VEL
LIN {X 0,Y 292.967,Z 449.248,A -85,B 0,C 180,E1 -16665.3,E2 -16665.3} C_VEL
LIN {X 0,Y 294.296,Z 442.17,A -85,B 0,C 180,E1 -16666.901,E2 -16666.901} C_VEL
LIN {X 0,Y 295.505,Z 434.45,A -85,B 0,C 180,E1 -16668.368,E2 -16668.368} C_VEL
LIN {X 0,Y 296.93,Z 425.923,A -85,B 0,C 180,E1 -16669.711,E2 -16669.711} C_VEL
LIN {X 0,Y 298.608,Z 415.63,A -85,B 0,C 180,E1 -16671.034,E2 -16671.034} C_VEL
LIN {X 0,Y 300.23,Z 403.225,A -85,B 0,C 180,E1 -16672.267,E2 -16672.267} C_VEL
LIN {X 0,Y 301.511,Z 392.421,A -85,B 0,C 180,E1 -16673.072,E2 -16673.072} C_VEL
LIN {X 0,Y 302.383,Z 382.494,A -85,B 0,C 180,E1 -16673.636,E2 -16673.636} C_VEL
LIN {X 0,Y 303.011,Z 372.639,A -85,B 0,C 180,E1 -16674.038,E2 -16674.038} C_VEL
LIN {X 0,Y 303.767,Z 347.209,A -85,B 0,C 180,E1 -16674.677,E2 -16674.677} C_VEL
LIN {X 0,Y 304.575,Z 310.036,A -85,B 0,C 180,E1 -16675.554,E2 -16675.554} C_VEL
LIN {X 0,Y 300.716,Z 288.338,A -85,B 0,C 180,E1 -16676.468,E2 -16676.468} C_VEL
LIN {X 0,Y 296.112,Z 267.954,A -85,B 0,C 180,E1 -16677.452,E2 -16677.452} C_VEL
LIN {X 0,Y 295.242,Z 265.243,A -85,B 0,C 180,E1 -16677.663,E2 -16677.663} C_VEL
LIN {X 0,Y 294.863,Z 263.02,A -85,B 0,C 180,E1 -16678.47,E2 -16678.47} C_VEL
LIN {X 0,Y 293.4,Z 255.171,A -85,B 0,C 180,E1 -16681.801,E2 -16681.801} C_VEL
LIN {X 0,Y 291.407,Z 245.723,A -85,B 0,C 180,E1 -16686.005,E2 -16686.005} C_VEL
LIN {X 0,Y 291.389,Z 245.662,A -85,B 0,C 180,E1 -16689.483,E2 -16689.483} C_VEL
LIN {X 0,Y 291.312,Z 245.7,A -85,B 0,C 180,E1 -16693.633,E2 -16693.633} C_VEL
LIN {X 0,Y 291.322,Z 245.698,A -85,B 0,C 180,E1 -16697.507,E2 -16697.507} C_VEL
LIN {X 0,Y 291.364,Z 245.682,A -85,B 0,C 180,E1 -16701.159,E2 -16701.159} C_VEL
LIN {X 0,Y 291.362,Z 245.678,A -85,B 0,C 180,E1 -16704.625,E2 -16704.625} C_VEL
LIN {X 0,Y 291.372,Z 245.685,A -85,B 0,C 180,E1 -16707.95,E2 -16707.95} C_VEL
LIN {X 0,Y 291.374,Z 245.678,A -85,B 0,C 180,E1 -16711.157,E2 -16711.157} C_VEL
LIN {X 0,Y 291.412,Z 245.663,A -85,B 0,C 180,E1 -16714.271,E2 -16714.271} C_VEL
LIN {X 0,Y 291.381,Z 245.688,A -85,B 0,C 180,E1 -16717.299,E2 -16717.299} C_VEL
LIN {X 0,Y 291.459,Z 245.65,A -85,B 0,C 180,E1 -16720.269,E2 -16720.269} C_VEL
LIN {X 0,Y 291.515,Z 245.665,A -85,B 0,C 180,E1 -16724.652,E2 -16724.652} C_VEL
LIN {X 0,Y 291.529,Z 245.642,A -85,B 0,C 180,E1 -16728.88,E2 -16728.88} C_VEL
LIN {X 0,Y 291.663,Z 245.623,A -85,B 0,C 180,E1 -16731.686,E2 -16731.686} C_VEL
LIN {X 0,Y 291.612,Z 245.657,A -85,B 0,C 180,E1 -16734.467,E2 -16734.467} C_VEL
LIN {X 0,Y 291.888,Z 245.598,A -85,B 0,C 180,E1 -16738.62,E2 -16738.62} C_VEL
LIN {X 0,Y 291.888,Z 245.593,A -85,B 0,C 180,E1 -16741.379,E2 -16741.379} C_VEL
LIN {X 0,Y 291.734,Z 245.636,A -85,B 0,C 180,E1 -16746.917,E2 -16746.917} C_VEL
LIN {X 0,Y 291.574,Z 245.626,A -85,B 0,C 180,E1 -16749.713,E2 -16749.713} C_VEL
LIN {X 0,Y 291.521,Z 245.669,A -85,B 0,C 180,E1 -16753.95,E2 -16753.95} C_VEL
LIN {X 0,Y 291.485,Z 245.663,A -85,B 0,C 180,E1 -16756.817,E2 -16756.817} C_VEL
LIN {X 0,Y 291.449,Z 245.649,A -85,B 0,C 180,E1 -16759.874,E2 -16759.874} C_VEL
LIN {X 0,Y 291.38,Z 245.688,A -85,B 0,C 180,E1 -16764.206,E2 -16764.206} C_VEL
LIN {X 0,Y 291.414,Z 245.655,A -85,B 0,C 180,E1 -16767.271,E2 -16767.271} C_VEL
LIN {X 0,Y 291.335,Z 245.696,A -85,B 0,C 180,E1 -16770.436,E2 -16770.436} C_VEL
LIN {X 0,Y 291.342,Z 245.676,A -85,B 0,C 180,E1 -16773.698,E2 -16773.698} C_VEL
LIN {X 0,Y 291.401,Z 245.687,A -85,B 0,C 180,E1 -16777.261,E2 -16777.261} C_VEL
LIN {X 0,Y 291.399,Z 245.669,A -85,B 0,C 180,E1 -16780.63,E2 -16780.63} C_VEL
LIN {X 0,Y 291.35,Z 245.688,A -85,B 0,C 180,E1 -16784.389,E2 -16784.389} C_VEL
LIN {X 0,Y 291.33,Z 245.642,A -85,B 0,C 180,E1 -16788.402,E2 -16788.402} C_VEL
LIN {X 0,Y 291.376,Z 245.686,A -85,B 0,C 180,E1 -16791.162,E2 -16791.162} C_VEL
LIN {X 0,Y 291.381,Z 245.657,A -85,B 0,C 180,E1 -16794.629,E2 -16794.629} C_VEL
LIN {X 0,Y 291.367,Z 245.691,A -85,B 0,C 180,E1 -16797.95,E2 -16797.95} C_VEL
LIN {X 0,Y 291.423,Z 245.829,A -85,B 0,C 180,E1 -16801.615,E2 -16801.615} C_VEL
LIN {X 0,Y 291.701,Z 246.892,A -85,B 0,C 180,E1 -16801.89,E2 -16801.89} C_VEL
LIN {X 0,Y 297.972,Z 258.644,A -85,B 0,C 180,E1 -16802.867,E2 -16802.867} C_VEL
LIN {X 0,Y 305.562,Z 269.338,A -85,B 0,C 180,E1 -16803.894,E2 -16803.894} C_VEL
LIN {X 0,Y 312.908,Z 277.767,A -85,B 0,C 180,E1 -16804.929,E2 -16804.929} C_VEL
LIN {X 0,Y 318.862,Z 284.205,A -85,B 0,C 180,E1 -16805.858,E2 -16805.858} C_VEL
LIN {X 0,Y 324.491,Z 290.173,A -85,B 0,C 180,E1 -16806.844,E2 -16806.844} C_VEL
LIN {X 0,Y 331.284,Z 296.914,A -85,B 0,C 180,E1 -16808.14,E2 -16808.14} C_VEL
LIN {X 0,Y 339.137,Z 304.329,A -85,B 0,C 180,E1 -16809.78,E2 -16809.78} C_VEL
LIN {X 0,Y 346.399,Z 310.791,A -85,B 0,C 180,E1 -16811.454,E2 -16811.454} C_VEL
LIN {X 0,Y 350.843,Z 314.392,A -85,B 0,C 180,E1 -16812.554,E2 -16812.554} C_VEL
LIN {X 0,Y 356.232,Z 319.009,A -85,B 0,C 180,E1 -16814.015,E2 -16814.015} C_VEL
LIN {X 0,Y 360.801,Z 322.485,A -85,B 0,C 180,E1 -16815.365,E2 -16815.365} C_VEL
LIN {X 0,Y 365.507,Z 326.379,A -85,B 0,C 180,E1 -16816.91,E2 -16816.91} C_VEL
LIN {X 0,Y 369.811,Z 329.163,A -85,B 0,C 180,E1 -16818.497,E2 -16818.497} C_VEL
LIN {X 0,Y 372.051,Z 330.69,A -85,B 0,C 180,E1 -16819.425,E2 -16819.425} C_VEL
LIN {X 0,Y 375.289,Z 333.586,A -85,B 0,C 180,E1 -16820.977,E2 -16820.977} C_VEL
LIN {X 0,Y 378.309,Z 335.709,A -85,B 0,C 180,E1 -16822.689,E2 -16822.689} C_VEL
LIN {X 0,Y 380.768,Z 337.069,A -85,B 0,C 180,E1 -16824.439,E2 -16824.439} C_VEL
LIN {X 0,Y 382.566,Z 337.76,A -85,B 0,C 180,E1 -16826.158,E2 -16826.158} C_VEL
LIN {X 0,Y 383.835,Z 338.319,A -85,B 0,C 180,E1 -16828.164,E2 -16828.164} C_VEL
LIN {X 0,Y 384.216,Z 338.461,A -85,B 0,C 180,E1 -16830,E2 -16830} C_VEL
LIN {X 0,Y 383.918,Z 338.383,A -85,B 0,C 180,E1 -16831.573,E2 -16831.573} C_VEL
LIN {X 0,Y 383.105,Z 337.908,A -85,B 0,C 180,E1 -16833.155,E2 -16833.155} C_VEL
LIN {X 0,Y 381.391,Z 337.38,A -85,B 0,C 180,E1 -16835.012,E2 -16835.012} C_VEL
LIN {X 0,Y 378.868,Z 336.055,A -85,B 0,C 180,E1 -16836.944,E2 -16836.944} C_VEL
LIN {X 0,Y 375.589,Z 333.826,A -85,B 0,C 180,E1 -16838.862,E2 -16838.862} C_VEL
LIN {X 0,Y 371.866,Z 330.528,A -85,B 0,C 180,E1 -16840.658,E2 -16840.658} C_VEL
LIN {X 0,Y 368.455,Z 328.357,A -85,B 0,C 180,E1 -16842.021,E2 -16842.021} C_VEL
LIN {X 0,Y 363.775,Z 325.048,A -85,B 0,C 180,E1 -16843.676,E2 -16843.676} C_VEL
LIN {X 0,Y 357.883,Z 320.163,A -85,B 0,C 180,E1 -16845.522,E2 -16845.522} C_VEL
LIN {X 0,Y 352.322,Z 315.811,A -85,B 0,C 180,E1 -16847.059,E2 -16847.059} C_VEL
LIN {X 0,Y 347.75,Z 311.821,A -85,B 0,C 180,E1 -16848.222,E2 -16848.222} C_VEL
LIN {X 0,Y 342.312,Z 307.203,A -85,B 0,C 180,E1 -16849.501,E2 -16849.501} C_VEL
LIN {X 0,Y 334.941,Z 300.519,A -85,B 0,C 180,E1 -16851.107,E2 -16851.107} C_VEL
LIN {X 0,Y 326.868,Z 292.55,A -85,B 0,C 180,E1 -16852.716,E2 -16852.716} C_VEL
LIN {X 0,Y 320.475,Z 286.027,A -85,B 0,C 180,E1 -16853.863,E2 -16853.863} C_VEL
LIN {X 0,Y 312.858,Z 277.733,A -85,B 0,C 180,E1 -16855.08,E2 -16855.08} C_VEL
LIN {X 0,Y 304.937,Z 268.505,A -85,B 0,C 180,E1 -16856.194,E2 -16856.194} C_VEL
LIN {X 0,Y 297.624,Z 258.048,A -85,B 0,C 180,E1 -16857.184,E2 -16857.184} C_VEL
LIN {X 0,Y 291.646,Z 246.783,A -85,B 0,C 180,E1 -16858.131,E2 -16858.131} C_VEL
LIN {X 0,Y 291.407,Z 245.751,A -85,B 0,C 180,E1 -16858.451,E2 -16858.451} C_VEL
LIN {X 0,Y 291.339,Z 245.687,A -85,B 0,C 180,E1 -16862.404,E2 -16862.404} C_VEL
LIN {X 0,Y 291.381,Z 245.657,A -85,B 0,C 180,E1 -16865.371,E2 -16865.371} C_VEL
LIN {X 0,Y 291.376,Z 245.686,A -85,B 0,C 180,E1 -16868.838,E2 -16868.838} C_VEL
LIN {X 0,Y 291.337,Z 245.642,A -85,B 0,C 180,E1 -16872.489,E2 -16872.489} C_VEL
LIN {X 0,Y 291.368,Z 245.693,A -85,B 0,C 180,E1 -16876.354,E2 -16876.354} C_VEL
LIN {X 0,Y 291.404,Z 245.676,A -85,B 0,C 180,E1 -16880.513,E2 -16880.513} C_VEL
LIN {X 0,Y 291.431,Z 245.683,A -85,B 0,C 180,E1 -16882.924,E2 -16882.924} C_VEL
LIN {X 0,Y 291.342,Z 245.676,A -85,B 0,C 180,E1 -16886.302,E2 -16886.302} C_VEL
LIN {X 0,Y 291.385,Z 245.683,A -85,B 0,C 180,E1 -16890.261,E2 -16890.261} C_VEL
LIN {X 0,Y 291.409,Z 245.669,A -85,B 0,C 180,E1 -16894.272,E2 -16894.272} C_VEL
LIN {X 0,Y 291.372,Z 245.691,A -85,B 0,C 180,E1 -16897.3,E2 -16897.3} C_VEL
LIN {X 0,Y 291.456,Z 245.647,A -85,B 0,C 180,E1 -16900.271,E2 -16900.271} C_VEL
LIN {X 0,Y 291.554,Z 245.665,A -85,B 0,C 180,E1 -16904.624,E2 -16904.624} C_VEL
LIN {X 0,Y 291.534,Z 245.639,A -85,B 0,C 180,E1 -16908.881,E2 -16908.881} C_VEL
LIN {X 0,Y 291.686,Z 245.624,A -85,B 0,C 180,E1 -16911.689,E2 -16911.689} C_VEL
LIN {X 0,Y 291.626,Z 245.657,A -85,B 0,C 180,E1 -16914.469,E2 -16914.469} C_VEL
LIN {X 0,Y 291.888,Z 245.593,A -85,B 0,C 180,E1 -16918.621,E2 -16918.621} C_VEL
LIN {X 0,Y 291.888,Z 245.598,A -85,B 0,C 180,E1 -16921.38,E2 -16921.38} C_VEL
LIN {X 0,Y 291.612,Z 245.657,A -85,B 0,C 180,E1 -16925.533,E2 -16925.533} C_VEL
LIN {X 0,Y 291.674,Z 245.615,A -85,B 0,C 180,E1 -16928.919,E2 -16928.919} C_VEL
LIN {X 0,Y 291.511,Z 245.668,A -85,B 0,C 180,E1 -16933.869,E2 -16933.869} C_VEL
LIN {X 0,Y 290.873,Z 245.752,A -85,B 0,C 180,E1 -16935.021,E2 -16935.021} C_VEL
LIN {X 0,Y 287.957,Z 246.099,A -85,B 0,C 180,E1 -16936.895,E2 -16936.895} C_VEL
LIN {X 0,Y 285.479,Z 246.392,A -85,B 0,C 180,E1 -16938.418,E2 -16938.418} C_VEL
LIN {X 0,Y 284.447,Z 246.522,A -85,B 0,C 180,E1 -16939.599,E2 -16939.599} C_VEL
LIN {X 0,Y 284.383,Z 246.534,A -85,B 0,C 180,E1 -16939.999,E2 -16939.999} C_VEL
LIN {X 0,Y 284.369,Z 246.559,A -85,B 0,C 180,E1 -16943.876,E2 -16943.876} C_VEL
LIN {X 0,Y 284.393,Z 246.531,A -85,B 0,C 180,E1 -16947.172,E2 -16947.172} C_VEL
LIN {X 0,Y 284.295,Z 246.57,A -85,B 0,C 180,E1 -16951.275,E2 -16951.275} C_VEL
LIN {X 0,Y 284.342,Z 246.551,A -85,B 0,C 180,E1 -16955.349,E2 -16955.349} C_VEL
LIN {X 0,Y 284.32,Z 246.566,A -85,B 0,C 180,E1 -16958.169,E2 -16958.169} C_VEL
LIN {X 0,Y 284.271,Z 246.575,A -85,B 0,C 180,E1 -16962.125,E2 -16962.125} C_VEL
LIN {X 0,Y 284.258,Z 246.578,A -85,B 0,C 180,E1 -16966.19,E2 -16966.19} C_VEL
LIN {X 0,Y 284.309,Z 246.54,A -85,B 0,C 180,E1 -16970.024,E2 -16970.024} C_VEL
LIN {X 0,Y 284.395,Z 246.706,A -85,B 0,C 180,E1 -16973.514,E2 -16973.514} C_VEL
LIN {X 0,Y 286.085,Z 254.951,A -85,B 0,C 180,E1 -16977.286,E2 -16977.286} C_VEL
LIN {X 0,Y 287.654,Z 262.807,A -85,B 0,C 180,E1 -16980.749,E2 -16980.749} C_VEL
LIN {X 0,Y 288.065,Z 265.081,A -85,B 0,C 180,E1 -16981.593,E2 -16981.593} C_VEL
LIN {X 0,Y 290.554,Z 272.093,A -85,B 0,C 180,E1 -16982.095,E2 -16982.095} C_VEL
LIN {X 0,Y 295.439,Z 295.278,A -85,B 0,C 180,E1 -16983.21,E2 -16983.21} C_VEL
LIN {X 0,Y 298.237,Z 311.426,A -85,B 0,C 180,E1 -16983.904,E2 -16983.904} C_VEL
LIN {X 0,Y 296.645,Z 371.115,A -85,B 0,C 180,E1 -16985.366,E2 -16985.366} C_VEL
LIN {X 0,Y 295.947,Z 381.427,A -85,B 0,C 180,E1 -16985.771,E2 -16985.771} C_VEL
LIN {X 0,Y 295.067,Z 390.939,A -85,B 0,C 180,E1 -16986.301,E2 -16986.301} C_VEL
LIN {X 0,Y 294.02,Z 400.012,A -85,B 0,C 180,E1 -16986.958,E2 -16986.958} C_VEL
LIN {X 0,Y 292.811,Z 409.143,A -85,B 0,C 180,E1 -16987.788,E2 -16987.788} C_VEL
LIN {X 0,Y 291.552,Z 418.139,A -85,B 0,C 180,E1 -16988.803,E2 -16988.803} C_VEL
LIN {X 0,Y 290.027,Z 426.863,A -85,B 0,C 180,E1 -16989.984,E2 -16989.984} C_VEL
LIN {X 0,Y 288.731,Z 434.256,A -85,B 0,C 180,E1 -16991.185,E2 -16991.185} C_VEL
LIN {X 0,Y 287.63,Z 441.293,A -85,B 0,C 180,E1 -16992.541,E2 -16992.541} C_VEL
LIN {X 0,Y 286.363,Z 447.678,A -85,B 0,C 180,E1 -16993.972,E2 -16993.972} C_VEL
LIN {X 0,Y 285.158,Z 454.216,A -85,B 0,C 180,E1 -16995.732,E2 -16995.732} C_VEL
LIN {X 0,Y 284.294,Z 458.716,A -85,B 0,C 180,E1 -16997.145,E2 -16997.145} C_VEL
LIN {X 0,Y 283.422,Z 464.211,A -85,B 0,C 180,E1 -16999.282,E2 -16999.282} C_VEL
LIN {X 0,Y 282.805,Z 468.538,A -85,B 0,C 180,E1 -17001.425,E2 -17001.425} C_VEL
LIN {X 0,Y 282.557,Z 470.907,A -85,B 0,C 180,E1 -17002.856,E2 -17002.856} C_VEL
LIN {X 0,Y 282.362,Z 473.137,A -85,B 0,C 180,E1 -17004.631,E2 -17004.631} C_VEL
LIN {X 0,Y 282.338,Z 475.159,A -85,B 0,C 180,E1 -17007.146,E2 -17007.146} C_VEL
LIN {X 0,Y 282.332,Z 475.749,A -85,B 0,C 180,E1 -17008.574,E2 -17008.574} C_VEL
LIN {X 0,Y 282.332,Z 475.749,A -85,B 0,C 180,E1 -17011.426,E2 -17011.426} C_VEL
LIN {X 0,Y 282.337,Z 475.159,A -85,B 0,C 180,E1 -17012.854,E2 -17012.854} C_VEL
